KUKA KRL program: cilindro.src, cilindro.dat

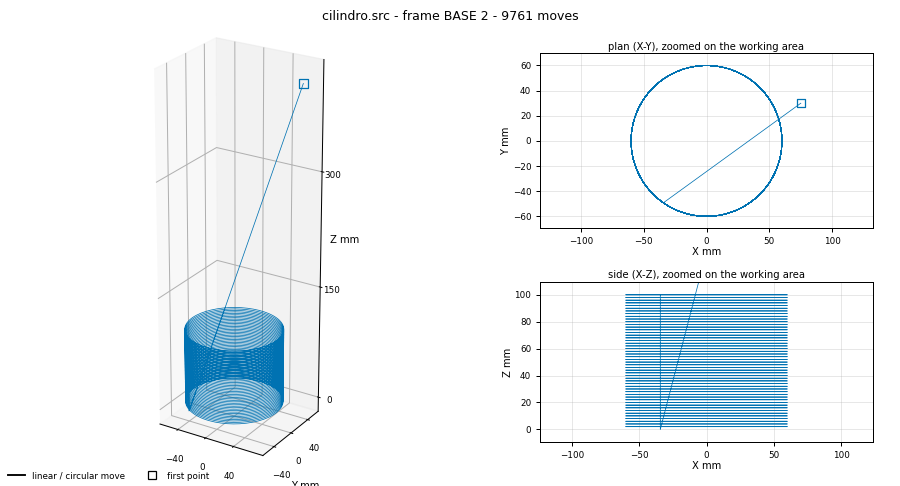
[picture p0: tool path of cilindro.src in frame BASE 2, 9761 of 9763 moves have a stored position in this frame; points joined in program order, loops and branches not executed]
--- cilindro.src ---
&ACCESS RVP
&PARAM TEMPLATE = C:\KRC\Roboter\Template\vorgabe
&PARAM EDITMASK = *
DEF cilindro( )
;FOLD INI;%{PE}%V3.2.0,%MKUKATPBASIS,%CINIT,%VCOMMON,%P
;FOLD BAS INI;%{E}%V3.2.0,%MKUKATPBASIS,%CINIT,%VINIT,%P
GLOBAL INTERRUPT DECL 3 WHEN $STOPMESS==TRUE DO IR_STOPM ( )
INTERRUPT ON 3
BAS (#INITMOV,0 )
;ENDFOLD (BAS INI)
;FOLD A20 INI;%{E}%V3.2.0,%MKUKATPA20,%CINIT,%VINIT,%P
IF ARC20==TRUE THEN
A20 (ARC_INI)
INTERRUPT DECL 6 WHEN $CYCFLAG[3]==FALSE DO A20(TECH_STOP2)
ENDIF
;ENDFOLD (A20 INI)
;FOLD A10 INI;%{E}%V3.2.0,%MKUKATPARC,%CINIT,%VINIT,%P
IF A10_OPTION==#ACTIVE THEN
INTERRUPT DECL 4 WHEN $CYCFLAG[2]==FALSE DO A10 (#APPL_ERROR)
INTERRUPT DECL 7 WHEN A_ARC_SWI==#ACTIVE DO A10 (#ARC_SEAM)
INTERRUPT DECL 5 WHEN A_FLY_ARC==TRUE DO A10 (#HPU_ARC)
INTERRUPT  ON 5
A10_INI ( )
ENDIF
;ENDFOLD (A10 INI)
;FOLD GRIPPER INI;%{E}%V3.2.0,%MKUKATPGRIPPER,%CINIT,%VINIT,%P
USER_GRP(0,DUMMY,DUMMY,GDEFAULT)
;ENDFOLD (GRIPPER INI)
;FOLD SPOT INI;%{E}%V3.2.0,%MKUKATPSPOT,%CINIT,%VINIT,%P
USERSPOT(#INIT)
;ENDFOLD (SPOT INI)
;FOLD TOUCHSENSE INI;%{E}%V3.2.0,%MKUKATPTS,%CINIT,%VINIT,%P
IF H70_OPTION THEN
INTERRUPT DECL 15 WHEN $MEAS_PULSE[TOUCH_I[TOUCH_ACTIVE].IN_NR] DO H70 (6,CD0 )
INTERRUPT DECL 16 WHEN $ZERO_MOVE DO H70 (7,CD0 )
INTERRUPT DECL 17 WHEN $TECHPAR_C[FG_TOUCH,8]>0.5 DO H70 (8,CD0)
H70 (1,CD0 )
ENDIF
;ENDFOLD (TOUCHSENSE INI)
;FOLD USER INI;%{E}%V3.2.0,%MKUKATPUSER,%CINIT,%VINIT,%P
;Make your modifications here
;ENDFOLD (USER INI)
;ENDFOLD (INI)
; SPEED PTP FOR AXIS
$VEL_AXIS[1] = 15
$VEL_AXIS[2] = 15
$VEL_AXIS[3] = 15
$VEL_AXIS[4] = 15
$VEL_AXIS[5] = 15
$VEL_AXIS[6] = 15
;SMOOTHNESS
$APO.CDIS = 2
;ADVANCE
$ADVANCE = 3
;SET TOOL AND BASE
$TOOL = TOOL_DATA[3]
$BASE = BASE_DATA[2]
;HOME
;FOLD PTP HOME Vel=10% DEFAULT
$BWDSTART=FALSE
$H_POS=XHOME
PDAT_ACT=PDEFAULT
FDAT_ACT=FHOME
BAS(#PTP_DAT )
BAS (#VEL_PTP,10 )
PTP XHOME
;ENDFOLD
;USER PROGRAM
;SPEED $VEL.CP
$VEL.CP=0.025
; OUT[TEMP] = 200
; OUT[vent] = 1
; OUT[RPM] = 25
$OUT[1] = TRUE
WAIT SEC 20
$OUT[1] = FALSE
; USER POSES CALLS
PTP {X 75, Y 30, Z 420, A 0, B 90, C 0}
; USER POSES CALLS
LIN {X -34.33, Y -49.21, Z 0.0, A 0, B 90, C 0} C_DIS
WAIT SEC 3
LIN {X -34.33, Y -49.21, Z 2.0, A 0, B 90, C 0} C_DIS
$OUT[1] = TRUE
WAIT SEC 0.8
LIN {X -34.33, Y -49.21, Z 2.0, A 0, B 90, C 0} C_DIS
LIN {X -34.33, Y -49.21, Z 2.0, A 0, B 90, C 0} C_DIS
LIN {X -31.1, Y -51.31, Z 2.0, A 0, B 90, C 0} C_DIS
LIN {X -27.75, Y -53.2, Z 2.0, A 0, B 90, C 0} C_DIS
LIN {X -24.29, Y -54.86, Z 2.0, A 0, B 90, C 0} C_DIS
LIN {X -20.72, Y -56.31, Z 2.0, A 0, B 90, C 0} C_DIS
LIN {X -17.07, Y -57.52, Z 2.0, A 0, B 90, C 0} C_DIS
LIN {X -13.35, Y -58.5, Z 2.0, A 0, B 90, C 0} C_DIS
LIN {X -9.58, Y -59.23, Z 2.0, A 0, B 90, C 0} C_DIS
LIN {X -5.76, Y -59.72, Z 2.0, A 0, B 90, C 0} C_DIS
LIN {X -1.92, Y -59.97, Z 2.0, A 0, B 90, C 0} C_DIS
LIN {X 1.92, Y -59.97, Z 2.0, A 0, B 90, C 0} C_DIS
LIN {X 5.76, Y -59.72, Z 2.0, A 0, B 90, C 0} C_DIS
LIN {X 9.58, Y -59.23, Z 2.0, A 0, B 90, C 0} C_DIS
LIN {X 13.35, Y -58.5, Z 2.0, A 0, B 90, C 0} C_DIS
LIN {X 17.07, Y -57.52, Z 2.0, A 0, B 90, C 0} C_DIS
LIN {X 20.72, Y -56.31, Z 2.0, A 0, B 90, C 0} C_DIS
LIN {X 24.29, Y -54.86, Z 2.0, A 0, B 90, C 0} C_DIS
LIN {X 27.75, Y -53.2, Z 2.0, A 0, B 90, C 0} C_DIS
LIN {X 31.1, Y -51.31, Z 2.0, A 0, B 90, C 0} C_DIS
LIN {X 34.33, Y -49.21, Z 2.0, A 0, B 90, C 0} C_DIS
LIN {X 37.41, Y -46.91, Z 2.0, A 0, B 90, C 0} C_DIS
LIN {X 40.34, Y -44.42, Z 2.0, A 0, B 90, C 0} C_DIS
LIN {X 43.1, Y -41.74, Z 2.0, A 0, B 90, C 0} C_DIS
LIN {X 45.69, Y -38.89, Z 2.0, A 0, B 90, C 0} C_DIS
LIN {X 48.08, Y -35.89, Z 2.0, A 0, B 90, C 0} C_DIS
LIN {X 50.29, Y -32.73, Z 2.0, A 0, B 90, C 0} C_DIS
LIN {X 52.28, Y -29.44, Z 2.0, A 0, B 90, C 0} C_DIS
LIN {X 54.06, Y -26.03, Z 2.0, A 0, B 90, C 0} C_DIS
LIN {X 55.62, Y -22.52, Z 2.0, A 0, B 90, C 0} C_DIS
LIN {X 56.94, Y -18.91, Z 2.0, A 0, B 90, C 0} C_DIS
LIN {X 58.04, Y -15.22, Z 2.0, A 0, B 90, C 0} C_DIS
LIN {X 58.89, Y -11.47, Z 2.0, A 0, B 90, C 0} C_DIS
LIN {X 59.51, Y -7.67, Z 2.0, A 0, B 90, C 0} C_DIS
LIN {X 59.88, Y -3.84, Z 2.0, A 0, B 90, C 0} C_DIS
LIN {X 60.0, Y 0.0, Z 2.0, A 0, B 90, C 0} C_DIS
LIN {X 59.88, Y 3.84, Z 2.0, A 0, B 90, C 0} C_DIS
LIN {X 59.51, Y 7.67, Z 2.0, A 0, B 90, C 0} C_DIS
LIN {X 58.89, Y 11.47, Z 2.0, A 0, B 90, C 0} C_DIS
LIN {X 58.04, Y 15.22, Z 2.0, A 0, B 90, C 0} C_DIS
LIN {X 56.94, Y 18.91, Z 2.0, A 0, B 90, C 0} C_DIS
LIN {X 55.62, Y 22.52, Z 2.0, A 0, B 90, C 0} C_DIS
LIN {X 54.06, Y 26.03, Z 2.0, A 0, B 90, C 0} C_DIS
LIN {X 52.28, Y 29.44, Z 2.0, A 0, B 90, C 0} C_DIS
LIN {X 50.29, Y 32.73, Z 2.0, A 0, B 90, C 0} C_DIS
LIN {X 48.08, Y 35.89, Z 2.0, A 0, B 90, C 0} C_DIS
LIN {X 45.69, Y 38.89, Z 2.0, A 0, B 90, C 0} C_DIS
LIN {X 43.1, Y 41.74, Z 2.0, A 0, B 90, C 0} C_DIS
LIN {X 40.34, Y 44.42, Z 2.0, A 0, B 90, C 0} C_DIS
LIN {X 37.41, Y 46.91, Z 2.0, A 0, B 90, C 0} C_DIS
LIN {X 34.33, Y 49.21, Z 2.0, A 0, B 90, C 0} C_DIS
LIN {X 31.1, Y 51.31, Z 2.0, A 0, B 90, C 0} C_DIS
LIN {X 27.75, Y 53.2, Z 2.0, A 0, B 90, C 0} C_DIS
LIN {X 24.29, Y 54.86, Z 2.0, A 0, B 90, C 0} C_DIS
LIN {X 20.72, Y 56.31, Z 2.0, A 0, B 90, C 0} C_DIS
LIN {X 17.07, Y 57.52, Z 2.0, A 0, B 90, C 0} C_DIS
LIN {X 13.35, Y 58.5, Z 2.0, A 0, B 90, C 0} C_DIS
LIN {X 9.58, Y 59.23, Z 2.0, A 0, B 90, C 0} C_DIS
LIN {X 5.76, Y 59.72, Z 2.0, A 0, B 90, C 0} C_DIS
LIN {X 1.92, Y 59.97, Z 2.0, A 0, B 90, C 0} C_DIS
LIN {X -1.92, Y 59.97, Z 2.0, A 0, B 90, C 0} C_DIS
LIN {X -5.76, Y 59.72, Z 2.0, A 0, B 90, C 0} C_DIS
LIN {X -9.58, Y 59.23, Z 2.0, A 0, B 90, C 0} C_DIS
LIN {X -13.35, Y 58.5, Z 2.0, A 0, B 90, C 0} C_DIS
LIN {X -17.07, Y 57.52, Z 2.0, A 0, B 90, C 0} C_DIS
LIN {X -20.72, Y 56.31, Z 2.0, A 0, B 90, C 0} C_DIS
LIN {X -24.29, Y 54.86, Z 2.0, A 0, B 90, C 0} C_DIS
LIN {X -27.75, Y 53.2, Z 2.0, A 0, B 90, C 0} C_DIS
LIN {X -31.1, Y 51.31, Z 2.0, A 0, B 90, C 0} C_DIS
LIN {X -34.33, Y 49.21, Z 2.0, A 0, B 90, C 0} C_DIS
LIN {X -37.41, Y 46.91, Z 2.0, A 0, B 90, C 0} C_DIS
LIN {X -40.34, Y 44.42, Z 2.0, A 0, B 90, C 0} C_DIS
LIN {X -43.1, Y 41.74, Z 2.0, A 0, B 90, C 0} C_DIS
LIN {X -45.69, Y 38.89, Z 2.0, A 0, B 90, C 0} C_DIS
LIN {X -48.08, Y 35.89, Z 2.0, A 0, B 90, C 0} C_DIS
LIN {X -50.29, Y 32.73, Z 2.0, A 0, B 90, C 0} C_DIS
LIN {X -52.28, Y 29.44, Z 2.0, A 0, B 90, C 0} C_DIS
LIN {X -54.06, Y 26.03, Z 2.0, A 0, B 90, C 0} C_DIS
LIN {X -55.62, Y 22.52, Z 2.0, A 0, B 90, C 0} C_DIS
LIN {X -56.94, Y 18.91, Z 2.0, A 0, B 90, C 0} C_DIS
LIN {X -58.04, Y 15.22, Z 2.0, A 0, B 90, C 0} C_DIS
LIN {X -58.89, Y 11.47, Z 2.0, A 0, B 90, C 0} C_DIS
LIN {X -59.51, Y 7.67, Z 2.0, A 0, B 90, C 0} C_DIS
LIN {X -59.88, Y 3.84, Z 2.0, A 0, B 90, C 0} C_DIS
LIN {X -60.0, Y -0.0, Z 2.0, A 0, B 90, C 0} C_DIS
LIN {X -59.88, Y -3.84, Z 2.0, A 0, B 90, C 0} C_DIS
LIN {X -59.51, Y -7.67, Z 2.0, A 0, B 90, C 0} C_DIS
LIN {X -58.89, Y -11.47, Z 2.0, A 0, B 90, C 0} C_DIS
LIN {X -58.04, Y -15.22, Z 2.0, A 0, B 90, C 0} C_DIS
LIN {X -56.94, Y -18.91, Z 2.0, A 0, B 90, C 0} C_DIS
LIN {X -55.62, Y -22.52, Z 2.0, A 0, B 90, C 0} C_DIS
LIN {X -54.06, Y -26.03, Z 2.0, A 0, B 90, C 0} C_DIS
LIN {X -52.28, Y -29.44, Z 2.0, A 0, B 90, C 0} C_DIS
LIN {X -50.29, Y -32.73, Z 2.0, A 0, B 90, C 0} C_DIS
LIN {X -48.08, Y -35.89, Z 2.0, A 0, B 90, C 0} C_DIS
LIN {X -45.69, Y -38.89, Z 2.0, A 0, B 90, C 0} C_DIS
LIN {X -43.1, Y -41.74, Z 2.0, A 0, B 90, C 0} C_DIS
LIN {X -40.34, Y -44.42, Z 2.0, A 0, B 90, C 0} C_DIS
LIN {X -37.41, Y -46.91, Z 2.0, A 0, B 90, C 0} C_DIS
LIN {X -37.13, Y -47.12, Z 2.0, A 0, B 90, C 0} C_DIS
$OUT[1] = FALSE

; END LAYER 0
LIN {X -34.33, Y -49.21, Z 2.0, A 0, B 90, C 0} C_DIS
WAIT SEC 3
LIN {X -34.33, Y -49.21, Z 4.0, A 0, B 90, C 0} C_DIS
$OUT[1] = TRUE
WAIT SEC 0.8
LIN {X -34.33, Y -49.21, Z 4.0, A 0, B 90, C 0} C_DIS
LIN {X -34.33, Y -49.21, Z 4.0, A 0, B 90, C 0} C_DIS
LIN {X -34.2, Y -49.29, Z 4.0, A 0, B 90, C 0} C_DIS
LIN {X -31.1, Y -51.31, Z 4.0, A 0, B 90, C 0} C_DIS
LIN {X -30.97, Y -51.38, Z 4.0, A 0, B 90, C 0} C_DIS
LIN {X -27.75, Y -53.2, Z 4.0, A 0, B 90, C 0} C_DIS
LIN {X -27.61, Y -53.26, Z 4.0, A 0, B 90, C 0} C_DIS
LIN {X -24.29, Y -54.86, Z 4.0, A 0, B 90, C 0} C_DIS
LIN {X -24.14, Y -54.92, Z 4.0, A 0, B 90, C 0} C_DIS
LIN {X -20.72, Y -56.31, Z 4.0, A 0, B 90, C 0} C_DIS
LIN {X -20.58, Y -56.36, Z 4.0, A 0, B 90, C 0} C_DIS
LIN {X -17.07, Y -57.52, Z 4.0, A 0, B 90, C 0} C_DIS
LIN {X -16.92, Y -57.56, Z 4.0, A 0, B 90, C 0} C_DIS
LIN {X -13.35, Y -58.5, Z 4.0, A 0, B 90, C 0} C_DIS
LIN {X -13.2, Y -58.53, Z 4.0, A 0, B 90, C 0} C_DIS
LIN {X -9.58, Y -59.23, Z 4.0, A 0, B 90, C 0} C_DIS
LIN {X -9.42, Y -59.25, Z 4.0, A 0, B 90, C 0} C_DIS
LIN {X -5.76, Y -59.72, Z 4.0, A 0, B 90, C 0} C_DIS
LIN {X -5.61, Y -59.73, Z 4.0, A 0, B 90, C 0} C_DIS
LIN {X -1.92, Y -59.97, Z 4.0, A 0, B 90, C 0} C_DIS
LIN {X -1.77, Y -59.97, Z 4.0, A 0, B 90, C 0} C_DIS
LIN {X 1.92, Y -59.97, Z 4.0, A 0, B 90, C 0} C_DIS
LIN {X 2.08, Y -59.96, Z 4.0, A 0, B 90, C 0} C_DIS
LIN {X 5.76, Y -59.72, Z 4.0, A 0, B 90, C 0} C_DIS
LIN {X 5.91, Y -59.7, Z 4.0, A 0, B 90, C 0} C_DIS
LIN {X 9.58, Y -59.23, Z 4.0, A 0, B 90, C 0} C_DIS
LIN {X 9.73, Y -59.2, Z 4.0, A 0, B 90, C 0} C_DIS
LIN {X 13.35, Y -58.5, Z 4.0, A 0, B 90, C 0} C_DIS
LIN {X 13.5, Y -58.46, Z 4.0, A 0, B 90, C 0} C_DIS
LIN {X 17.07, Y -57.52, Z 4.0, A 0, B 90, C 0} C_DIS
LIN {X 17.22, Y -57.47, Z 4.0, A 0, B 90, C 0} C_DIS
LIN {X 20.72, Y -56.31, Z 4.0, A 0, B 90, C 0} C_DIS
LIN {X 20.86, Y -56.25, Z 4.0, A 0, B 90, C 0} C_DIS
LIN {X 24.29, Y -54.86, Z 4.0, A 0, B 90, C 0} C_DIS
LIN {X 24.43, Y -54.8, Z 4.0, A 0, B 90, C 0} C_DIS
LIN {X 27.75, Y -53.2, Z 4.0, A 0, B 90, C 0} C_DIS
LIN {X 27.89, Y -53.12, Z 4.0, A 0, B 90, C 0} C_DIS
LIN {X 31.1, Y -51.31, Z 4.0, A 0, B 90, C 0} C_DIS
LIN {X 31.23, Y -51.22, Z 4.0, A 0, B 90, C 0} C_DIS
LIN {X 34.33, Y -49.21, Z 4.0, A 0, B 90, C 0} C_DIS
LIN {X 34.45, Y -49.12, Z 4.0, A 0, B 90, C 0} C_DIS
LIN {X 37.41, Y -46.91, Z 4.0, A 0, B 90, C 0} C_DIS
LIN {X 37.53, Y -46.81, Z 4.0, A 0, B 90, C 0} C_DIS
LIN {X 40.34, Y -44.42, Z 4.0, A 0, B 90, C 0} C_DIS
LIN {X 40.45, Y -44.31, Z 4.0, A 0, B 90, C 0} C_DIS
LIN {X 43.1, Y -41.74, Z 4.0, A 0, B 90, C 0} C_DIS
LIN {X 43.2, Y -41.63, Z 4.0, A 0, B 90, C 0} C_DIS
LIN {X 45.69, Y -38.89, Z 4.0, A 0, B 90, C 0} C_DIS
LIN {X 45.78, Y -38.77, Z 4.0, A 0, B 90, C 0} C_DIS
LIN {X 48.08, Y -35.89, Z 4.0, A 0, B 90, C 0} C_DIS
LIN {X 48.17, Y -35.76, Z 4.0, A 0, B 90, C 0} C_DIS
LIN {X 50.29, Y -32.73, Z 4.0, A 0, B 90, C 0} C_DIS
LIN {X 50.37, Y -32.6, Z 4.0, A 0, B 90, C 0} C_DIS
LIN {X 52.28, Y -29.44, Z 4.0, A 0, B 90, C 0} C_DIS
LIN {X 52.35, Y -29.31, Z 4.0, A 0, B 90, C 0} C_DIS
LIN {X 54.06, Y -26.03, Z 4.0, A 0, B 90, C 0} C_DIS
LIN {X 54.12, Y -25.89, Z 4.0, A 0, B 90, C 0} C_DIS
LIN {X 55.62, Y -22.52, Z 4.0, A 0, B 90, C 0} C_DIS
LIN {X 55.67, Y -22.37, Z 4.0, A 0, B 90, C 0} C_DIS
LIN {X 56.94, Y -18.91, Z 4.0, A 0, B 90, C 0} C_DIS
LIN {X 56.99, Y -18.76, Z 4.0, A 0, B 90, C 0} C_DIS
LIN {X 58.04, Y -15.22, Z 4.0, A 0, B 90, C 0} C_DIS
LIN {X 58.07, Y -15.07, Z 4.0, A 0, B 90, C 0} C_DIS
LIN {X 58.89, Y -11.47, Z 4.0, A 0, B 90, C 0} C_DIS
LIN {X 58.92, Y -11.32, Z 4.0, A 0, B 90, C 0} C_DIS
LIN {X 59.51, Y -7.67, Z 4.0, A 0, B 90, C 0} C_DIS
LIN {X 59.52, Y -7.52, Z 4.0, A 0, B 90, C 0} C_DIS
LIN {X 59.88, Y -3.84, Z 4.0, A 0, B 90, C 0} C_DIS
LIN {X 59.88, Y -3.69, Z 4.0, A 0, B 90, C 0} C_DIS
LIN {X 60.0, Y 0.0, Z 4.0, A 0, B 90, C 0} C_DIS
LIN {X 60.0, Y 0.15, Z 4.0, A 0, B 90, C 0} C_DIS
LIN {X 59.88, Y 3.84, Z 4.0, A 0, B 90, C 0} C_DIS
LIN {X 59.86, Y 4.0, Z 4.0, A 0, B 90, C 0} C_DIS
LIN {X 59.51, Y 7.67, Z 4.0, A 0, B 90, C 0} C_DIS
LIN {X 59.48, Y 7.82, Z 4.0, A 0, B 90, C 0} C_DIS
LIN {X 58.89, Y 11.47, Z 4.0, A 0, B 90, C 0} C_DIS
LIN {X 58.86, Y 11.62, Z 4.0, A 0, B 90, C 0} C_DIS
LIN {X 58.04, Y 15.22, Z 4.0, A 0, B 90, C 0} C_DIS
LIN {X 57.99, Y 15.37, Z 4.0, A 0, B 90, C 0} C_DIS
LIN {X 56.94, Y 18.91, Z 4.0, A 0, B 90, C 0} C_DIS
LIN {X 56.89, Y 19.05, Z 4.0, A 0, B 90, C 0} C_DIS
LIN {X 55.62, Y 22.52, Z 4.0, A 0, B 90, C 0} C_DIS
LIN {X 55.55, Y 22.66, Z 4.0, A 0, B 90, C 0} C_DIS
LIN {X 54.06, Y 26.03, Z 4.0, A 0, B 90, C 0} C_DIS
LIN {X 53.99, Y 26.17, Z 4.0, A 0, B 90, C 0} C_DIS
LIN {X 52.28, Y 29.44, Z 4.0, A 0, B 90, C 0} C_DIS
LIN {X 52.2, Y 29.57, Z 4.0, A 0, B 90, C 0} C_DIS
LIN {X 50.29, Y 32.73, Z 4.0, A 0, B 90, C 0} C_DIS
LIN {X 50.2, Y 32.86, Z 4.0, A 0, B 90, C 0} C_DIS
LIN {X 48.08, Y 35.89, Z 4.0, A 0, B 90, C 0} C_DIS
LIN {X 47.99, Y 36.01, Z 4.0, A 0, B 90, C 0} C_DIS
LIN {X 45.69, Y 38.89, Z 4.0, A 0, B 90, C 0} C_DIS
LIN {X 45.58, Y 39.01, Z 4.0, A 0, B 90, C 0} C_DIS
LIN {X 43.1, Y 41.74, Z 4.0, A 0, B 90, C 0} C_DIS
LIN {X 42.99, Y 41.85, Z 4.0, A 0, B 90, C 0} C_DIS
LIN {X 40.34, Y 44.42, Z 4.0, A 0, B 90, C 0} C_DIS
LIN {X 40.22, Y 44.52, Z 4.0, A 0, B 90, C 0} C_DIS
LIN {X 37.41, Y 46.91, Z 4.0, A 0, B 90, C 0} C_DIS
LIN {X 37.29, Y 47.0, Z 4.0, A 0, B 90, C 0} C_DIS
LIN {X 34.33, Y 49.21, Z 4.0, A 0, B 90, C 0} C_DIS
LIN {X 34.2, Y 49.29, Z 4.0, A 0, B 90, C 0} C_DIS
LIN {X 31.1, Y 51.31, Z 4.0, A 0, B 90, C 0} C_DIS
LIN {X 30.97, Y 51.38, Z 4.0, A 0, B 90, C 0} C_DIS
LIN {X 27.75, Y 53.2, Z 4.0, A 0, B 90, C 0} C_DIS
LIN {X 27.61, Y 53.26, Z 4.0, A 0, B 90, C 0} C_DIS
LIN {X 24.29, Y 54.86, Z 4.0, A 0, B 90, C 0} C_DIS
LIN {X 24.14, Y 54.92, Z 4.0, A 0, B 90, C 0} C_DIS
LIN {X 20.72, Y 56.31, Z 4.0, A 0, B 90, C 0} C_DIS
LIN {X 20.58, Y 56.36, Z 4.0, A 0, B 90, C 0} C_DIS
LIN {X 17.07, Y 57.52, Z 4.0, A 0, B 90, C 0} C_DIS
LIN {X 16.92, Y 57.56, Z 4.0, A 0, B 90, C 0} C_DIS
LIN {X 13.35, Y 58.5, Z 4.0, A 0, B 90, C 0} C_DIS
LIN {X 13.2, Y 58.53, Z 4.0, A 0, B 90, C 0} C_DIS
LIN {X 9.58, Y 59.23, Z 4.0, A 0, B 90, C 0} C_DIS
LIN {X 9.42, Y 59.25, Z 4.0, A 0, B 90, C 0} C_DIS
LIN {X 5.76, Y 59.72, Z 4.0, A 0, B 90, C 0} C_DIS
LIN {X 5.61, Y 59.73, Z 4.0, A 0, B 90, C 0} C_DIS
LIN {X 1.92, Y 59.97, Z 4.0, A 0, B 90, C 0} C_DIS
LIN {X 1.77, Y 59.97, Z 4.0, A 0, B 90, C 0} C_DIS
LIN {X -1.92, Y 59.97, Z 4.0, A 0, B 90, C 0} C_DIS
LIN {X -2.08, Y 59.96, Z 4.0, A 0, B 90, C 0} C_DIS
LIN {X -5.76, Y 59.72, Z 4.0, A 0, B 90, C 0} C_DIS
LIN {X -5.91, Y 59.7, Z 4.0, A 0, B 90, C 0} C_DIS
LIN {X -9.58, Y 59.23, Z 4.0, A 0, B 90, C 0} C_DIS
LIN {X -9.73, Y 59.2, Z 4.0, A 0, B 90, C 0} C_DIS
LIN {X -13.35, Y 58.5, Z 4.0, A 0, B 90, C 0} C_DIS
LIN {X -13.5, Y 58.46, Z 4.0, A 0, B 90, C 0} C_DIS
LIN {X -17.07, Y 57.52, Z 4.0, A 0, B 90, C 0} C_DIS
LIN {X -17.22, Y 57.47, Z 4.0, A 0, B 90, C 0} C_DIS
LIN {X -20.72, Y 56.31, Z 4.0, A 0, B 90, C 0} C_DIS
LIN {X -20.86, Y 56.25, Z 4.0, A 0, B 90, C 0} C_DIS
LIN {X -24.29, Y 54.86, Z 4.0, A 0, B 90, C 0} C_DIS
LIN {X -24.43, Y 54.8, Z 4.0, A 0, B 90, C 0} C_DIS
LIN {X -27.75, Y 53.2, Z 4.0, A 0, B 90, C 0} C_DIS
LIN {X -27.89, Y 53.12, Z 4.0, A 0, B 90, C 0} C_DIS
LIN {X -31.1, Y 51.31, Z 4.0, A 0, B 90, C 0} C_DIS
LIN {X -31.23, Y 51.22, Z 4.0, A 0, B 90, C 0} C_DIS
LIN {X -34.33, Y 49.21, Z 4.0, A 0, B 90, C 0} C_DIS
LIN {X -34.45, Y 49.12, Z 4.0, A 0, B 90, C 0} C_DIS
LIN {X -37.41, Y 46.91, Z 4.0, A 0, B 90, C 0} C_DIS
LIN {X -37.53, Y 46.81, Z 4.0, A 0, B 90, C 0} C_DIS
LIN {X -40.34, Y 44.42, Z 4.0, A 0, B 90, C 0} C_DIS
LIN {X -40.45, Y 44.31, Z 4.0, A 0, B 90, C 0} C_DIS
LIN {X -43.1, Y 41.74, Z 4.0, A 0, B 90, C 0} C_DIS
LIN {X -43.2, Y 41.63, Z 4.0, A 0, B 90, C 0} C_DIS
LIN {X -45.69, Y 38.89, Z 4.0, A 0, B 90, C 0} C_DIS
LIN {X -45.78, Y 38.77, Z 4.0, A 0, B 90, C 0} C_DIS
LIN {X -48.08, Y 35.89, Z 4.0, A 0, B 90, C 0} C_DIS
LIN {X -48.17, Y 35.76, Z 4.0, A 0, B 90, C 0} C_DIS
LIN {X -50.29, Y 32.73, Z 4.0, A 0, B 90, C 0} C_DIS
LIN {X -50.37, Y 32.6, Z 4.0, A 0, B 90, C 0} C_DIS
LIN {X -52.28, Y 29.44, Z 4.0, A 0, B 90, C 0} C_DIS
LIN {X -52.35, Y 29.31, Z 4.0, A 0, B 90, C 0} C_DIS
LIN {X -54.06, Y 26.03, Z 4.0, A 0, B 90, C 0} C_DIS
LIN {X -54.12, Y 25.89, Z 4.0, A 0, B 90, C 0} C_DIS
LIN {X -55.62, Y 22.52, Z 4.0, A 0, B 90, C 0} C_DIS
LIN {X -55.67, Y 22.37, Z 4.0, A 0, B 90, C 0} C_DIS
LIN {X -56.94, Y 18.91, Z 4.0, A 0, B 90, C 0} C_DIS
LIN {X -56.99, Y 18.76, Z 4.0, A 0, B 90, C 0} C_DIS
LIN {X -58.04, Y 15.22, Z 4.0, A 0, B 90, C 0} C_DIS
LIN {X -58.07, Y 15.07, Z 4.0, A 0, B 90, C 0} C_DIS
LIN {X -58.89, Y 11.47, Z 4.0, A 0, B 90, C 0} C_DIS
LIN {X -58.92, Y 11.32, Z 4.0, A 0, B 90, C 0} C_DIS
LIN {X -59.51, Y 7.67, Z 4.0, A 0, B 90, C 0} C_DIS
LIN {X -59.52, Y 7.52, Z 4.0, A 0, B 90, C 0} C_DIS
LIN {X -59.88, Y 3.84, Z 4.0, A 0, B 90, C 0} C_DIS
LIN {X -59.88, Y 3.69, Z 4.0, A 0, B 90, C 0} C_DIS
LIN {X -60.0, Y -0.0, Z 4.0, A 0, B 90, C 0} C_DIS
LIN {X -60.0, Y -0.15, Z 4.0, A 0, B 90, C 0} C_DIS
LIN {X -59.88, Y -3.84, Z 4.0, A 0, B 90, C 0} C_DIS
LIN {X -59.86, Y -4.0, Z 4.0, A 0, B 90, C 0} C_DIS
LIN {X -59.51, Y -7.67, Z 4.0, A 0, B 90, C 0} C_DIS
LIN {X -59.48, Y -7.82, Z 4.0, A 0, B 90, C 0} C_DIS
LIN {X -58.89, Y -11.47, Z 4.0, A 0, B 90, C 0} C_DIS
LIN {X -58.86, Y -11.62, Z 4.0, A 0, B 90, C 0} C_DIS
LIN {X -58.04, Y -15.22, Z 4.0, A 0, B 90, C 0} C_DIS
LIN {X -57.99, Y -15.37, Z 4.0, A 0, B 90, C 0} C_DIS
LIN {X -56.94, Y -18.91, Z 4.0, A 0, B 90, C 0} C_DIS
LIN {X -56.89, Y -19.05, Z 4.0, A 0, B 90, C 0} C_DIS
LIN {X -55.62, Y -22.52, Z 4.0, A 0, B 90, C 0} C_DIS
LIN {X -55.55, Y -22.66, Z 4.0, A 0, B 90, C 0} C_DIS
LIN {X -54.06, Y -26.03, Z 4.0, A 0, B 90, C 0} C_DIS
LIN {X -53.99, Y -26.17, Z 4.0, A 0, B 90, C 0} C_DIS
LIN {X -52.28, Y -29.44, Z 4.0, A 0, B 90, C 0} C_DIS
LIN {X -52.2, Y -29.57, Z 4.0, A 0, B 90, C 0} C_DIS
LIN {X -50.29, Y -32.73, Z 4.0, A 0, B 90, C 0} C_DIS
LIN {X -50.2, Y -32.86, Z 4.0, A 0, B 90, C 0} C_DIS
LIN {X -48.08, Y -35.89, Z 4.0, A 0, B 90, C 0} C_DIS
LIN {X -47.99, Y -36.01, Z 4.0, A 0, B 90, C 0} C_DIS
LIN {X -45.69, Y -38.89, Z 4.0, A 0, B 90, C 0} C_DIS
LIN {X -45.58, Y -39.01, Z 4.0, A 0, B 90, C 0} C_DIS
LIN {X -43.1, Y -41.74, Z 4.0, A 0, B 90, C 0} C_DIS
LIN {X -42.99, Y -41.85, Z 4.0, A 0, B 90, C 0} C_DIS
LIN {X -40.34, Y -44.42, Z 4.0, A 0, B 90, C 0} C_DIS
LIN {X -40.22, Y -44.52, Z 4.0, A 0, B 90, C 0} C_DIS
LIN {X -37.41, Y -46.91, Z 4.0, A 0, B 90, C 0} C_DIS
LIN {X -37.29, Y -47.0, Z 4.0, A 0, B 90, C 0} C_DIS
LIN {X -37.13, Y -47.12, Z 4.0, A 0, B 90, C 0} C_DIS
$OUT[1] = FALSE

; END LAYER 1
LIN {X -34.33, Y -49.21, Z 4.0, A 0, B 90, C 0} C_DIS
WAIT SEC 3
LIN {X -34.33, Y -49.21, Z 6.0, A 0, B 90, C 0} C_DIS
$OUT[1] = TRUE
WAIT SEC 0.8
LIN {X -34.33, Y -49.21, Z 6.0, A 0, B 90, C 0} C_DIS
LIN {X -34.33, Y -49.21, Z 6.0, A 0, B 90, C 0} C_DIS
LIN {X -34.07, Y -49.38, Z 6.0, A 0, B 90, C 0} C_DIS
LIN {X -31.1, Y -51.31, Z 6.0, A 0, B 90, C 0} C_DIS
LIN {X -30.84, Y -51.46, Z 6.0, A 0, B 90, C 0} C_DIS
LIN {X -27.75, Y -53.2, Z 6.0, A 0, B 90, C 0} C_DIS
LIN {X -27.48, Y -53.33, Z 6.0, A 0, B 90, C 0} C_DIS
LIN {X -24.29, Y -54.86, Z 6.0, A 0, B 90, C 0} C_DIS
LIN {X -24.0, Y -54.98, Z 6.0, A 0, B 90, C 0} C_DIS
LIN {X -20.72, Y -56.31, Z 6.0, A 0, B 90, C 0} C_DIS
LIN {X -20.43, Y -56.41, Z 6.0, A 0, B 90, C 0} C_DIS
LIN {X -17.07, Y -57.52, Z 6.0, A 0, B 90, C 0} C_DIS
LIN {X -16.77, Y -57.6, Z 6.0, A 0, B 90, C 0} C_DIS
LIN {X -13.35, Y -58.5, Z 6.0, A 0, B 90, C 0} C_DIS
LIN {X -13.05, Y -58.55, Z 6.0, A 0, B 90, C 0} C_DIS
LIN {X -9.58, Y -59.23, Z 6.0, A 0, B 90, C 0} C_DIS
LIN {X -9.27, Y -59.27, Z 6.0, A 0, B 90, C 0} C_DIS
LIN {X -5.76, Y -59.72, Z 6.0, A 0, B 90, C 0} C_DIS
LIN {X -5.45, Y -59.74, Z 6.0, A 0, B 90, C 0} C_DIS
LIN {X -1.92, Y -59.97, Z 6.0, A 0, B 90, C 0} C_DIS
LIN {X -1.62, Y -59.97, Z 6.0, A 0, B 90, C 0} C_DIS
LIN {X 1.92, Y -59.97, Z 6.0, A 0, B 90, C 0} C_DIS
LIN {X 2.23, Y -59.95, Z 6.0, A 0, B 90, C 0} C_DIS
LIN {X 5.76, Y -59.72, Z 6.0, A 0, B 90, C 0} C_DIS
LIN {X 6.07, Y -59.68, Z 6.0, A 0, B 90, C 0} C_DIS
LIN {X 9.58, Y -59.23, Z 6.0, A 0, B 90, C 0} C_DIS
LIN {X 9.88, Y -59.17, Z 6.0, A 0, B 90, C 0} C_DIS
LIN {X 13.35, Y -58.5, Z 6.0, A 0, B 90, C 0} C_DIS
LIN {X 13.65, Y -58.42, Z 6.0, A 0, B 90, C 0} C_DIS
LIN {X 17.07, Y -57.52, Z 6.0, A 0, B 90, C 0} C_DIS
LIN {X 17.36, Y -57.42, Z 6.0, A 0, B 90, C 0} C_DIS
LIN {X 20.72, Y -56.31, Z 6.0, A 0, B 90, C 0} C_DIS
LIN {X 21.01, Y -56.19, Z 6.0, A 0, B 90, C 0} C_DIS
LIN {X 24.29, Y -54.86, Z 6.0, A 0, B 90, C 0} C_DIS
LIN {X 24.56, Y -54.73, Z 6.0, A 0, B 90, C 0} C_DIS
LIN {X 27.75, Y -53.2, Z 6.0, A 0, B 90, C 0} C_DIS
LIN {X 28.02, Y -53.04, Z 6.0, A 0, B 90, C 0} C_DIS
LIN {X 31.1, Y -51.31, Z 6.0, A 0, B 90, C 0} C_DIS
LIN {X 31.36, Y -51.14, Z 6.0, A 0, B 90, C 0} C_DIS
LIN {X 34.33, Y -49.21, Z 6.0, A 0, B 90, C 0} C_DIS
LIN {X 34.57, Y -49.03, Z 6.0, A 0, B 90, C 0} C_DIS
LIN {X 37.41, Y -46.91, Z 6.0, A 0, B 90, C 0} C_DIS
LIN {X 37.64, Y -46.71, Z 6.0, A 0, B 90, C 0} C_DIS
LIN {X 40.34, Y -44.42, Z 6.0, A 0, B 90, C 0} C_DIS
LIN {X 40.56, Y -44.2, Z 6.0, A 0, B 90, C 0} C_DIS
LIN {X 43.1, Y -41.74, Z 6.0, A 0, B 90, C 0} C_DIS
LIN {X 43.31, Y -41.51, Z 6.0, A 0, B 90, C 0} C_DIS
LIN {X 45.69, Y -38.89, Z 6.0, A 0, B 90, C 0} C_DIS
LIN {X 45.88, Y -38.65, Z 6.0, A 0, B 90, C 0} C_DIS
LIN {X 48.08, Y -35.89, Z 6.0, A 0, B 90, C 0} C_DIS
LIN {X 48.26, Y -35.63, Z 6.0, A 0, B 90, C 0} C_DIS
LIN {X 50.29, Y -32.73, Z 6.0, A 0, B 90, C 0} C_DIS
LIN {X 50.44, Y -32.47, Z 6.0, A 0, B 90, C 0} C_DIS
LIN {X 52.28, Y -29.44, Z 6.0, A 0, B 90, C 0} C_DIS
LIN {X 52.42, Y -29.17, Z 6.0, A 0, B 90, C 0} C_DIS
LIN {X 54.06, Y -26.03, Z 6.0, A 0, B 90, C 0} C_DIS
LIN {X 54.18, Y -25.75, Z 6.0, A 0, B 90, C 0} C_DIS
LIN {X 55.62, Y -22.52, Z 6.0, A 0, B 90, C 0} C_DIS
LIN {X 55.72, Y -22.23, Z 6.0, A 0, B 90, C 0} C_DIS
LIN {X 56.94, Y -18.91, Z 6.0, A 0, B 90, C 0} C_DIS
LIN {X 57.03, Y -18.61, Z 6.0, A 0, B 90, C 0} C_DIS
LIN {X 58.04, Y -15.22, Z 6.0, A 0, B 90, C 0} C_DIS
LIN {X 58.11, Y -14.92, Z 6.0, A 0, B 90, C 0} C_DIS
LIN {X 58.89, Y -11.47, Z 6.0, A 0, B 90, C 0} C_DIS
LIN {X 58.94, Y -11.17, Z 6.0, A 0, B 90, C 0} C_DIS
LIN {X 59.51, Y -7.67, Z 6.0, A 0, B 90, C 0} C_DIS
LIN {X 59.54, Y -7.37, Z 6.0, A 0, B 90, C 0} C_DIS
LIN {X 59.88, Y -3.84, Z 6.0, A 0, B 90, C 0} C_DIS
LIN {X 59.89, Y -3.54, Z 6.0, A 0, B 90, C 0} C_DIS
LIN {X 60.0, Y 0.0, Z 6.0, A 0, B 90, C 0} C_DIS
LIN {X 59.99, Y 0.31, Z 6.0, A 0, B 90, C 0} C_DIS
LIN {X 59.88, Y 3.84, Z 6.0, A 0, B 90, C 0} C_DIS
LIN {X 59.85, Y 4.15, Z 6.0, A 0, B 90, C 0} C_DIS
LIN {X 59.51, Y 7.67, Z 6.0, A 0, B 90, C 0} C_DIS
LIN {X 59.46, Y 7.98, Z 6.0, A 0, B 90, C 0} C_DIS
LIN {X 58.89, Y 11.47, Z 6.0, A 0, B 90, C 0} C_DIS
LIN {X 58.83, Y 11.77, Z 6.0, A 0, B 90, C 0} C_DIS
LIN {X 58.04, Y 15.22, Z 6.0, A 0, B 90, C 0} C_DIS
LIN {X 57.95, Y 15.51, Z 6.0, A 0, B 90, C 0} C_DIS
LIN {X 56.94, Y 18.91, Z 6.0, A 0, B 90, C 0} C_DIS
LIN {X 56.84, Y 19.2, Z 6.0, A 0, B 90, C 0} C_DIS
LIN {X 55.62, Y 22.52, Z 6.0, A 0, B 90, C 0} C_DIS
LIN {X 55.49, Y 22.8, Z 6.0, A 0, B 90, C 0} C_DIS
LIN {X 54.06, Y 26.03, Z 6.0, A 0, B 90, C 0} C_DIS
LIN {X 53.92, Y 26.31, Z 6.0, A 0, B 90, C 0} C_DIS
LIN {X 52.28, Y 29.44, Z 6.0, A 0, B 90, C 0} C_DIS
LIN {X 52.12, Y 29.71, Z 6.0, A 0, B 90, C 0} C_DIS
LIN {X 50.29, Y 32.73, Z 6.0, A 0, B 90, C 0} C_DIS
LIN {X 50.11, Y 32.98, Z 6.0, A 0, B 90, C 0} C_DIS
LIN {X 48.08, Y 35.89, Z 6.0, A 0, B 90, C 0} C_DIS
LIN {X 47.89, Y 36.13, Z 6.0, A 0, B 90, C 0} C_DIS
LIN {X 45.69, Y 38.89, Z 6.0, A 0, B 90, C 0} C_DIS
LIN {X 45.48, Y 39.12, Z 6.0, A 0, B 90, C 0} C_DIS
LIN {X 43.1, Y 41.74, Z 6.0, A 0, B 90, C 0} C_DIS
LIN {X 42.88, Y 41.96, Z 6.0, A 0, B 90, C 0} C_DIS
LIN {X 40.34, Y 44.42, Z 6.0, A 0, B 90, C 0} C_DIS
LIN {X 40.1, Y 44.62, Z 6.0, A 0, B 90, C 0} C_DIS
LIN {X 37.41, Y 46.91, Z 6.0, A 0, B 90, C 0} C_DIS
LIN {X 37.16, Y 47.09, Z 6.0, A 0, B 90, C 0} C_DIS
LIN {X 34.33, Y 49.21, Z 6.0, A 0, B 90, C 0} C_DIS
LIN {X 34.07, Y 49.38, Z 6.0, A 0, B 90, C 0} C_DIS
LIN {X 31.1, Y 51.31, Z 6.0, A 0, B 90, C 0} C_DIS
LIN {X 30.84, Y 51.46, Z 6.0, A 0, B 90, C 0} C_DIS
LIN {X 27.75, Y 53.2, Z 6.0, A 0, B 90, C 0} C_DIS
LIN {X 27.48, Y 53.33, Z 6.0, A 0, B 90, C 0} C_DIS
LIN {X 24.29, Y 54.86, Z 6.0, A 0, B 90, C 0} C_DIS
LIN {X 24.0, Y 54.98, Z 6.0, A 0, B 90, C 0} C_DIS
LIN {X 20.72, Y 56.31, Z 6.0, A 0, B 90, C 0} C_DIS
LIN {X 20.43, Y 56.41, Z 6.0, A 0, B 90, C 0} C_DIS
LIN {X 17.07, Y 57.52, Z 6.0, A 0, B 90, C 0} C_DIS
LIN {X 16.77, Y 57.6, Z 6.0, A 0, B 90, C 0} C_DIS
LIN {X 13.35, Y 58.5, Z 6.0, A 0, B 90, C 0} C_DIS
LIN {X 13.05, Y 58.55, Z 6.0, A 0, B 90, C 0} C_DIS
LIN {X 9.58, Y 59.23, Z 6.0, A 0, B 90, C 0} C_DIS
LIN {X 9.27, Y 59.27, Z 6.0, A 0, B 90, C 0} C_DIS
LIN {X 5.76, Y 59.72, Z 6.0, A 0, B 90, C 0} C_DIS
LIN {X 5.45, Y 59.74, Z 6.0, A 0, B 90, C 0} C_DIS
LIN {X 1.92, Y 59.97, Z 6.0, A 0, B 90, C 0} C_DIS
LIN {X 1.62, Y 59.97, Z 6.0, A 0, B 90, C 0} C_DIS
LIN {X -1.92, Y 59.97, Z 6.0, A 0, B 90, C 0} C_DIS
LIN {X -2.23, Y 59.95, Z 6.0, A 0, B 90, C 0} C_DIS
LIN {X -5.76, Y 59.72, Z 6.0, A 0, B 90, C 0} C_DIS
LIN {X -6.07, Y 59.68, Z 6.0, A 0, B 90, C 0} C_DIS
LIN {X -9.58, Y 59.23, Z 6.0, A 0, B 90, C 0} C_DIS
LIN {X -9.88, Y 59.17, Z 6.0, A 0, B 90, C 0} C_DIS
LIN {X -13.35, Y 58.5, Z 6.0, A 0, B 90, C 0} C_DIS
LIN {X -13.65, Y 58.42, Z 6.0, A 0, B 90, C 0} C_DIS
LIN {X -17.07, Y 57.52, Z 6.0, A 0, B 90, C 0} C_DIS
LIN {X -17.36, Y 57.42, Z 6.0, A 0, B 90, C 0} C_DIS
LIN {X -20.72, Y 56.31, Z 6.0, A 0, B 90, C 0} C_DIS
LIN {X -21.01, Y 56.19, Z 6.0, A 0, B 90, C 0} C_DIS
LIN {X -24.29, Y 54.86, Z 6.0, A 0, B 90, C 0} C_DIS
LIN {X -24.56, Y 54.73, Z 6.0, A 0, B 90, C 0} C_DIS
LIN {X -27.75, Y 53.2, Z 6.0, A 0, B 90, C 0} C_DIS
LIN {X -28.02, Y 53.04, Z 6.0, A 0, B 90, C 0} C_DIS
LIN {X -31.1, Y 51.31, Z 6.0, A 0, B 90, C 0} C_DIS
LIN {X -31.36, Y 51.14, Z 6.0, A 0, B 90, C 0} C_DIS
LIN {X -34.33, Y 49.21, Z 6.0, A 0, B 90, C 0} C_DIS
LIN {X -34.57, Y 49.03, Z 6.0, A 0, B 90, C 0} C_DIS
LIN {X -37.41, Y 46.91, Z 6.0, A 0, B 90, C 0} C_DIS
LIN {X -37.64, Y 46.71, Z 6.0, A 0, B 90, C 0} C_DIS
LIN {X -40.34, Y 44.42, Z 6.0, A 0, B 90, C 0} C_DIS
LIN {X -40.56, Y 44.2, Z 6.0, A 0, B 90, C 0} C_DIS
LIN {X -43.1, Y 41.74, Z 6.0, A 0, B 90, C 0} C_DIS
LIN {X -43.31, Y 41.51, Z 6.0, A 0, B 90, C 0} C_DIS
LIN {X -45.69, Y 38.89, Z 6.0, A 0, B 90, C 0} C_DIS
LIN {X -45.88, Y 38.65, Z 6.0, A 0, B 90, C 0} C_DIS
LIN {X -48.08, Y 35.89, Z 6.0, A 0, B 90, C 0} C_DIS
LIN {X -48.26, Y 35.63, Z 6.0, A 0, B 90, C 0} C_DIS
LIN {X -50.29, Y 32.73, Z 6.0, A 0, B 90, C 0} C_DIS
LIN {X -50.44, Y 32.47, Z 6.0, A 0, B 90, C 0} C_DIS
LIN {X -52.28, Y 29.44, Z 6.0, A 0, B 90, C 0} C_DIS
LIN {X -52.42, Y 29.17, Z 6.0, A 0, B 90, C 0} C_DIS
LIN {X -54.06, Y 26.03, Z 6.0, A 0, B 90, C 0} C_DIS
LIN {X -54.18, Y 25.75, Z 6.0, A 0, B 90, C 0} C_DIS
LIN {X -55.62, Y 22.52, Z 6.0, A 0, B 90, C 0} C_DIS
LIN {X -55.72, Y 22.23, Z 6.0, A 0, B 90, C 0} C_DIS
LIN {X -56.94, Y 18.91, Z 6.0, A 0, B 90, C 0} C_DIS
LIN {X -57.03, Y 18.61, Z 6.0, A 0, B 90, C 0} C_DIS
LIN {X -58.04, Y 15.22, Z 6.0, A 0, B 90, C 0} C_DIS
LIN {X -58.11, Y 14.92, Z 6.0, A 0, B 90, C 0} C_DIS
LIN {X -58.89, Y 11.47, Z 6.0, A 0, B 90, C 0} C_DIS
LIN {X -58.94, Y 11.17, Z 6.0, A 0, B 90, C 0} C_DIS
LIN {X -59.51, Y 7.67, Z 6.0, A 0, B 90, C 0} C_DIS
LIN {X -59.54, Y 7.37, Z 6.0, A 0, B 90, C 0} C_DIS
LIN {X -59.88, Y 3.84, Z 6.0, A 0, B 90, C 0} C_DIS
LIN {X -59.89, Y 3.54, Z 6.0, A 0, B 90, C 0} C_DIS
LIN {X -60.0, Y -0.0, Z 6.0, A 0, B 90, C 0} C_DIS
LIN {X -59.99, Y -0.31, Z 6.0, A 0, B 90, C 0} C_DIS
LIN {X -59.88, Y -3.84, Z 6.0, A 0, B 90, C 0} C_DIS
LIN {X -59.85, Y -4.15, Z 6.0, A 0, B 90, C 0} C_DIS
LIN {X -59.51, Y -7.67, Z 6.0, A 0, B 90, C 0} C_DIS
LIN {X -59.46, Y -7.98, Z 6.0, A 0, B 90, C 0} C_DIS
LIN {X -58.89, Y -11.47, Z 6.0, A 0, B 90, C 0} C_DIS
LIN {X -58.83, Y -11.77, Z 6.0, A 0, B 90, C 0} C_DIS
LIN {X -58.04, Y -15.22, Z 6.0, A 0, B 90, C 0} C_DIS
LIN {X -57.95, Y -15.51, Z 6.0, A 0, B 90, C 0} C_DIS
LIN {X -56.94, Y -18.91, Z 6.0, A 0, B 90, C 0} C_DIS
LIN {X -56.84, Y -19.2, Z 6.0, A 0, B 90, C 0} C_DIS
LIN {X -55.62, Y -22.52, Z 6.0, A 0, B 90, C 0} C_DIS
LIN {X -55.49, Y -22.8, Z 6.0, A 0, B 90, C 0} C_DIS
LIN {X -54.06, Y -26.03, Z 6.0, A 0, B 90, C 0} C_DIS
LIN {X -53.92, Y -26.31, Z 6.0, A 0, B 90, C 0} C_DIS
LIN {X -52.28, Y -29.44, Z 6.0, A 0, B 90, C 0} C_DIS
LIN {X -52.12, Y -29.71, Z 6.0, A 0, B 90, C 0} C_DIS
LIN {X -50.29, Y -32.73, Z 6.0, A 0, B 90, C 0} C_DIS
LIN {X -50.11, Y -32.98, Z 6.0, A 0, B 90, C 0} C_DIS
LIN {X -48.08, Y -35.89, Z 6.0, A 0, B 90, C 0} C_DIS
LIN {X -47.89, Y -36.13, Z 6.0, A 0, B 90, C 0} C_DIS
LIN {X -45.69, Y -38.89, Z 6.0, A 0, B 90, C 0} C_DIS
LIN {X -45.48, Y -39.12, Z 6.0, A 0, B 90, C 0} C_DIS
LIN {X -43.1, Y -41.74, Z 6.0, A 0, B 90, C 0} C_DIS
LIN {X -42.88, Y -41.96, Z 6.0, A 0, B 90, C 0} C_DIS
LIN {X -40.34, Y -44.42, Z 6.0, A 0, B 90, C 0} C_DIS
LIN {X -40.1, Y -44.62, Z 6.0, A 0, B 90, C 0} C_DIS
LIN {X -37.41, Y -46.91, Z 6.0, A 0, B 90, C 0} C_DIS
LIN {X -37.16, Y -47.09, Z 6.0, A 0, B 90, C 0} C_DIS
LIN {X -37.13, Y -47.11, Z 6.0, A 0, B 90, C 0} C_DIS
$OUT[1] = FALSE

; END LAYER 2
LIN {X -34.33, Y -49.21, Z 6.0, A 0, B 90, C 0} C_DIS
WAIT SEC 3
LIN {X -34.33, Y -49.21, Z 8.0, A 0, B 90, C 0} C_DIS
$OUT[1] = TRUE
WAIT SEC 0.8
LIN {X -34.33, Y -49.21, Z 8.0, A 0, B 90, C 0} C_DIS
LIN {X -34.33, Y -49.21, Z 8.0, A 0, B 90, C 0} C_DIS
LIN {X -33.94, Y -49.46, Z 8.0, A 0, B 90, C 0} C_DIS
LIN {X -31.1, Y -51.31, Z 8.0, A 0, B 90, C 0} C_DIS
LIN {X -30.7, Y -51.54, Z 8.0, A 0, B 90, C 0} C_DIS
LIN {X -27.75, Y -53.2, Z 8.0, A 0, B 90, C 0} C_DIS
LIN {X -27.34, Y -53.4, Z 8.0, A 0, B 90, C 0} C_DIS
LIN {X -24.29, Y -54.86, Z 8.0, A 0, B 90, C 0} C_DIS
LIN {X -23.86, Y -55.04, Z 8.0, A 0, B 90, C 0} C_DIS
LIN {X -20.72, Y -56.31, Z 8.0, A 0, B 90, C 0} C_DIS
LIN {X -20.28, Y -56.45, Z 8.0, A 0, B 90, C 0} C_DIS
LIN {X -17.07, Y -57.52, Z 8.0, A 0, B 90, C 0} C_DIS
LIN {X -16.63, Y -57.64, Z 8.0, A 0, B 90, C 0} C_DIS
LIN {X -13.35, Y -58.5, Z 8.0, A 0, B 90, C 0} C_DIS
LIN {X -12.9, Y -58.58, Z 8.0, A 0, B 90, C 0} C_DIS
LIN {X -9.58, Y -59.23, Z 8.0, A 0, B 90, C 0} C_DIS
LIN {X -9.12, Y -59.29, Z 8.0, A 0, B 90, C 0} C_DIS
LIN {X -5.76, Y -59.72, Z 8.0, A 0, B 90, C 0} C_DIS
LIN {X -5.3, Y -59.75, Z 8.0, A 0, B 90, C 0} C_DIS
LIN {X -1.92, Y -59.97, Z 8.0, A 0, B 90, C 0} C_DIS
LIN {X -1.46, Y -59.97, Z 8.0, A 0, B 90, C 0} C_DIS
LIN {X 1.92, Y -59.97, Z 8.0, A 0, B 90, C 0} C_DIS
LIN {X 2.38, Y -59.94, Z 8.0, A 0, B 90, C 0} C_DIS
LIN {X 5.76, Y -59.72, Z 8.0, A 0, B 90, C 0} C_DIS
LIN {X 6.22, Y -59.66, Z 8.0, A 0, B 90, C 0} C_DIS
LIN {X 9.58, Y -59.23, Z 8.0, A 0, B 90, C 0} C_DIS
LIN {X 10.03, Y -59.14, Z 8.0, A 0, B 90, C 0} C_DIS
LIN {X 13.35, Y -58.5, Z 8.0, A 0, B 90, C 0} C_DIS
LIN {X 13.8, Y -58.38, Z 8.0, A 0, B 90, C 0} C_DIS
LIN {X 17.07, Y -57.52, Z 8.0, A 0, B 90, C 0} C_DIS
LIN {X 17.51, Y -57.37, Z 8.0, A 0, B 90, C 0} C_DIS
LIN {X 20.72, Y -56.31, Z 8.0, A 0, B 90, C 0} C_DIS
LIN {X 21.15, Y -56.13, Z 8.0, A 0, B 90, C 0} C_DIS
LIN {X 24.29, Y -54.86, Z 8.0, A 0, B 90, C 0} C_DIS
LIN {X 24.7, Y -54.66, Z 8.0, A 0, B 90, C 0} C_DIS
LIN {X 27.75, Y -53.2, Z 8.0, A 0, B 90, C 0} C_DIS
LIN {X 28.15, Y -52.97, Z 8.0, A 0, B 90, C 0} C_DIS
LIN {X 31.1, Y -51.31, Z 8.0, A 0, B 90, C 0} C_DIS
LIN {X 31.49, Y -51.06, Z 8.0, A 0, B 90, C 0} C_DIS
LIN {X 34.33, Y -49.21, Z 8.0, A 0, B 90, C 0} C_DIS
LIN {X 34.7, Y -48.93, Z 8.0, A 0, B 90, C 0} C_DIS
LIN {X 37.41, Y -46.91, Z 8.0, A 0, B 90, C 0} C_DIS
LIN {X 37.76, Y -46.61, Z 8.0, A 0, B 90, C 0} C_DIS
LIN {X 40.34, Y -44.42, Z 8.0, A 0, B 90, C 0} C_DIS
LIN {X 40.67, Y -44.1, Z 8.0, A 0, B 90, C 0} C_DIS
LIN {X 43.1, Y -41.74, Z 8.0, A 0, B 90, C 0} C_DIS
LIN {X 43.41, Y -41.4, Z 8.0, A 0, B 90, C 0} C_DIS
LIN {X 45.69, Y -38.89, Z 8.0, A 0, B 90, C 0} C_DIS
LIN {X 45.97, Y -38.53, Z 8.0, A 0, B 90, C 0} C_DIS
LIN {X 48.08, Y -35.89, Z 8.0, A 0, B 90, C 0} C_DIS
LIN {X 48.35, Y -35.51, Z 8.0, A 0, B 90, C 0} C_DIS
LIN {X 50.29, Y -32.73, Z 8.0, A 0, B 90, C 0} C_DIS
LIN {X 50.52, Y -32.34, Z 8.0, A 0, B 90, C 0} C_DIS
LIN {X 52.28, Y -29.44, Z 8.0, A 0, B 90, C 0} C_DIS
LIN {X 52.49, Y -29.03, Z 8.0, A 0, B 90, C 0} C_DIS
LIN {X 54.06, Y -26.03, Z 8.0, A 0, B 90, C 0} C_DIS
LIN {X 54.24, Y -25.61, Z 8.0, A 0, B 90, C 0} C_DIS
LIN {X 55.62, Y -22.52, Z 8.0, A 0, B 90, C 0} C_DIS
LIN {X 55.77, Y -22.08, Z 8.0, A 0, B 90, C 0} C_DIS
LIN {X 56.94, Y -18.91, Z 8.0, A 0, B 90, C 0} C_DIS
LIN {X 57.07, Y -18.46, Z 8.0, A 0, B 90, C 0} C_DIS
LIN {X 58.04, Y -15.22, Z 8.0, A 0, B 90, C 0} C_DIS
LIN {X 58.14, Y -14.77, Z 8.0, A 0, B 90, C 0} C_DIS
LIN {X 58.89, Y -11.47, Z 8.0, A 0, B 90, C 0} C_DIS
LIN {X 58.97, Y -11.01, Z 8.0, A 0, B 90, C 0} C_DIS
LIN {X 59.51, Y -7.67, Z 8.0, A 0, B 90, C 0} C_DIS
LIN {X 59.55, Y -7.21, Z 8.0, A 0, B 90, C 0} C_DIS
LIN {X 59.88, Y -3.84, Z 8.0, A 0, B 90, C 0} C_DIS
LIN {X 59.89, Y -3.38, Z 8.0, A 0, B 90, C 0} C_DIS
LIN {X 60.0, Y 0.0, Z 8.0, A 0, B 90, C 0} C_DIS
LIN {X 59.99, Y 0.46, Z 8.0, A 0, B 90, C 0} C_DIS
LIN {X 59.88, Y 3.84, Z 8.0, A 0, B 90, C 0} C_DIS
LIN {X 59.83, Y 4.3, Z 8.0, A 0, B 90, C 0} C_DIS
LIN {X 59.51, Y 7.67, Z 8.0, A 0, B 90, C 0} C_DIS
LIN {X 59.43, Y 8.13, Z 8.0, A 0, B 90, C 0} C_DIS
LIN {X 58.89, Y 11.47, Z 8.0, A 0, B 90, C 0} C_DIS
LIN {X 58.79, Y 11.92, Z 8.0, A 0, B 90, C 0} C_DIS
LIN {X 58.04, Y 15.22, Z 8.0, A 0, B 90, C 0} C_DIS
LIN {X 57.91, Y 15.66, Z 8.0, A 0, B 90, C 0} C_DIS
LIN {X 56.94, Y 18.91, Z 8.0, A 0, B 90, C 0} C_DIS
LIN {X 56.78, Y 19.34, Z 8.0, A 0, B 90, C 0} C_DIS
LIN {X 55.62, Y 22.52, Z 8.0, A 0, B 90, C 0} C_DIS
LIN {X 55.43, Y 22.94, Z 8.0, A 0, B 90, C 0} C_DIS
LIN {X 54.06, Y 26.03, Z 8.0, A 0, B 90, C 0} C_DIS
LIN {X 53.84, Y 26.44, Z 8.0, A 0, B 90, C 0} C_DIS
LIN {X 52.28, Y 29.44, Z 8.0, A 0, B 90, C 0} C_DIS
LIN {X 52.04, Y 29.84, Z 8.0, A 0, B 90, C 0} C_DIS
LIN {X 50.29, Y 32.73, Z 8.0, A 0, B 90, C 0} C_DIS
LIN {X 50.02, Y 33.11, Z 8.0, A 0, B 90, C 0} C_DIS
LIN {X 48.08, Y 35.89, Z 8.0, A 0, B 90, C 0} C_DIS
LIN {X 47.8, Y 36.25, Z 8.0, A 0, B 90, C 0} C_DIS
LIN {X 45.69, Y 38.89, Z 8.0, A 0, B 90, C 0} C_DIS
LIN {X 45.38, Y 39.24, Z 8.0, A 0, B 90, C 0} C_DIS
LIN {X 43.1, Y 41.74, Z 8.0, A 0, B 90, C 0} C_DIS
LIN {X 42.77, Y 42.06, Z 8.0, A 0, B 90, C 0} C_DIS
LIN {X 40.34, Y 44.42, Z 8.0, A 0, B 90, C 0} C_DIS
LIN {X 39.99, Y 44.72, Z 8.0, A 0, B 90, C 0} C_DIS
LIN {X 37.41, Y 46.91, Z 8.0, A 0, B 90, C 0} C_DIS
LIN {X 37.04, Y 47.19, Z 8.0, A 0, B 90, C 0} C_DIS
LIN {X 34.33, Y 49.21, Z 8.0, A 0, B 90, C 0} C_DIS
LIN {X 33.94, Y 49.46, Z 8.0, A 0, B 90, C 0} C_DIS
LIN {X 31.1, Y 51.31, Z 8.0, A 0, B 90, C 0} C_DIS
LIN {X 30.7, Y 51.54, Z 8.0, A 0, B 90, C 0} C_DIS
LIN {X 27.75, Y 53.2, Z 8.0, A 0, B 90, C 0} C_DIS
LIN {X 27.34, Y 53.4, Z 8.0, A 0, B 90, C 0} C_DIS
LIN {X 24.29, Y 54.86, Z 8.0, A 0, B 90, C 0} C_DIS
LIN {X 23.86, Y 55.04, Z 8.0, A 0, B 90, C 0} C_DIS
LIN {X 20.72, Y 56.31, Z 8.0, A 0, B 90, C 0} C_DIS
LIN {X 20.28, Y 56.45, Z 8.0, A 0, B 90, C 0} C_DIS
LIN {X 17.07, Y 57.52, Z 8.0, A 0, B 90, C 0} C_DIS
LIN {X 16.63, Y 57.64, Z 8.0, A 0, B 90, C 0} C_DIS
LIN {X 13.35, Y 58.5, Z 8.0, A 0, B 90, C 0} C_DIS
LIN {X 12.9, Y 58.58, Z 8.0, A 0, B 90, C 0} C_DIS
LIN {X 9.58, Y 59.23, Z 8.0, A 0, B 90, C 0} C_DIS
LIN {X 9.12, Y 59.29, Z 8.0, A 0, B 90, C 0} C_DIS
LIN {X 5.76, Y 59.72, Z 8.0, A 0, B 90, C 0} C_DIS
LIN {X 5.3, Y 59.75, Z 8.0, A 0, B 90, C 0} C_DIS
LIN {X 1.92, Y 59.97, Z 8.0, A 0, B 90, C 0} C_DIS
LIN {X 1.46, Y 59.97, Z 8.0, A 0, B 90, C 0} C_DIS
LIN {X -1.92, Y 59.97, Z 8.0, A 0, B 90, C 0} C_DIS
LIN {X -2.38, Y 59.94, Z 8.0, A 0, B 90, C 0} C_DIS
LIN {X -5.76, Y 59.72, Z 8.0, A 0, B 90, C 0} C_DIS
LIN {X -6.22, Y 59.66, Z 8.0, A 0, B 90, C 0} C_DIS
LIN {X -9.58, Y 59.23, Z 8.0, A 0, B 90, C 0} C_DIS
LIN {X -10.03, Y 59.14, Z 8.0, A 0, B 90, C 0} C_DIS
LIN {X -13.35, Y 58.5, Z 8.0, A 0, B 90, C 0} C_DIS
LIN {X -13.8, Y 58.38, Z 8.0, A 0, B 90, C 0} C_DIS
LIN {X -17.07, Y 57.52, Z 8.0, A 0, B 90, C 0} C_DIS
LIN {X -17.51, Y 57.37, Z 8.0, A 0, B 90, C 0} C_DIS
LIN {X -20.72, Y 56.31, Z 8.0, A 0, B 90, C 0} C_DIS
LIN {X -21.15, Y 56.13, Z 8.0, A 0, B 90, C 0} C_DIS
LIN {X -24.29, Y 54.86, Z 8.0, A 0, B 90, C 0} C_DIS
LIN {X -24.7, Y 54.66, Z 8.0, A 0, B 90, C 0} C_DIS
LIN {X -27.75, Y 53.2, Z 8.0, A 0, B 90, C 0} C_DIS
LIN {X -28.15, Y 52.97, Z 8.0, A 0, B 90, C 0} C_DIS
LIN {X -31.1, Y 51.31, Z 8.0, A 0, B 90, C 0} C_DIS
LIN {X -31.49, Y 51.06, Z 8.0, A 0, B 90, C 0} C_DIS
LIN {X -34.33, Y 49.21, Z 8.0, A 0, B 90, C 0} C_DIS
LIN {X -34.7, Y 48.93, Z 8.0, A 0, B 90, C 0} C_DIS
LIN {X -37.41, Y 46.91, Z 8.0, A 0, B 90, C 0} C_DIS
LIN {X -37.76, Y 46.61, Z 8.0, A 0, B 90, C 0} C_DIS
LIN {X -40.34, Y 44.42, Z 8.0, A 0, B 90, C 0} C_DIS
LIN {X -40.67, Y 44.1, Z 8.0, A 0, B 90, C 0} C_DIS
LIN {X -43.1, Y 41.74, Z 8.0, A 0, B 90, C 0} C_DIS
LIN {X -43.41, Y 41.4, Z 8.0, A 0, B 90, C 0} C_DIS
LIN {X -45.69, Y 38.89, Z 8.0, A 0, B 90, C 0} C_DIS
LIN {X -45.97, Y 38.53, Z 8.0, A 0, B 90, C 0} C_DIS
LIN {X -48.08, Y 35.89, Z 8.0, A 0, B 90, C 0} C_DIS
LIN {X -48.35, Y 35.51, Z 8.0, A 0, B 90, C 0} C_DIS
LIN {X -50.29, Y 32.73, Z 8.0, A 0, B 90, C 0} C_DIS
LIN {X -50.52, Y 32.34, Z 8.0, A 0, B 90, C 0} C_DIS
LIN {X -52.28, Y 29.44, Z 8.0, A 0, B 90, C 0} C_DIS
LIN {X -52.49, Y 29.03, Z 8.0, A 0, B 90, C 0} C_DIS
LIN {X -54.06, Y 26.03, Z 8.0, A 0, B 90, C 0} C_DIS
LIN {X -54.24, Y 25.61, Z 8.0, A 0, B 90, C 0} C_DIS
LIN {X -55.62, Y 22.52, Z 8.0, A 0, B 90, C 0} C_DIS
LIN {X -55.77, Y 22.08, Z 8.0, A 0, B 90, C 0} C_DIS
LIN {X -56.94, Y 18.91, Z 8.0, A 0, B 90, C 0} C_DIS
LIN {X -57.07, Y 18.46, Z 8.0, A 0, B 90, C 0} C_DIS
LIN {X -58.04, Y 15.22, Z 8.0, A 0, B 90, C 0} C_DIS
LIN {X -58.14, Y 14.77, Z 8.0, A 0, B 90, C 0} C_DIS
LIN {X -58.89, Y 11.47, Z 8.0, A 0, B 90, C 0} C_DIS
LIN {X -58.97, Y 11.01, Z 8.0, A 0, B 90, C 0} C_DIS
LIN {X -59.51, Y 7.67, Z 8.0, A 0, B 90, C 0} C_DIS
LIN {X -59.55, Y 7.21, Z 8.0, A 0, B 90, C 0} C_DIS
LIN {X -59.88, Y 3.84, Z 8.0, A 0, B 90, C 0} C_DIS
LIN {X -59.89, Y 3.38, Z 8.0, A 0, B 90, C 0} C_DIS
LIN {X -60.0, Y -0.0, Z 8.0, A 0, B 90, C 0} C_DIS
LIN {X -59.99, Y -0.46, Z 8.0, A 0, B 90, C 0} C_DIS
LIN {X -59.88, Y -3.84, Z 8.0, A 0, B 90, C 0} C_DIS
LIN {X -59.83, Y -4.3, Z 8.0, A 0, B 90, C 0} C_DIS
LIN {X -59.51, Y -7.67, Z 8.0, A 0, B 90, C 0} C_DIS
LIN {X -59.43, Y -8.13, Z 8.0, A 0, B 90, C 0} C_DIS
LIN {X -58.89, Y -11.47, Z 8.0, A 0, B 90, C 0} C_DIS
LIN {X -58.79, Y -11.92, Z 8.0, A 0, B 90, C 0} C_DIS
LIN {X -58.04, Y -15.22, Z 8.0, A 0, B 90, C 0} C_DIS
LIN {X -57.91, Y -15.66, Z 8.0, A 0, B 90, C 0} C_DIS
LIN {X -56.94, Y -18.91, Z 8.0, A 0, B 90, C 0} C_DIS
LIN {X -56.78, Y -19.34, Z 8.0, A 0, B 90, C 0} C_DIS
LIN {X -55.62, Y -22.52, Z 8.0, A 0, B 90, C 0} C_DIS
LIN {X -55.43, Y -22.94, Z 8.0, A 0, B 90, C 0} C_DIS
LIN {X -54.06, Y -26.03, Z 8.0, A 0, B 90, C 0} C_DIS
LIN {X -53.84, Y -26.44, Z 8.0, A 0, B 90, C 0} C_DIS
LIN {X -52.28, Y -29.44, Z 8.0, A 0, B 90, C 0} C_DIS
LIN {X -52.04, Y -29.84, Z 8.0, A 0, B 90, C 0} C_DIS
LIN {X -50.29, Y -32.73, Z 8.0, A 0, B 90, C 0} C_DIS
LIN {X -50.02, Y -33.11, Z 8.0, A 0, B 90, C 0} C_DIS
LIN {X -48.08, Y -35.89, Z 8.0, A 0, B 90, C 0} C_DIS
LIN {X -47.8, Y -36.25, Z 8.0, A 0, B 90, C 0} C_DIS
LIN {X -45.69, Y -38.89, Z 8.0, A 0, B 90, C 0} C_DIS
LIN {X -45.38, Y -39.24, Z 8.0, A 0, B 90, C 0} C_DIS
LIN {X -43.1, Y -41.74, Z 8.0, A 0, B 90, C 0} C_DIS
LIN {X -42.77, Y -42.06, Z 8.0, A 0, B 90, C 0} C_DIS
LIN {X -40.34, Y -44.42, Z 8.0, A 0, B 90, C 0} C_DIS
LIN {X -39.99, Y -44.72, Z 8.0, A 0, B 90, C 0} C_DIS
LIN {X -37.41, Y -46.91, Z 8.0, A 0, B 90, C 0} C_DIS
LIN {X -37.04, Y -47.19, Z 8.0, A 0, B 90, C 0} C_DIS
$OUT[1] = FALSE

; END LAYER 3
LIN {X -34.33, Y -49.21, Z 8.0, A 0, B 90, C 0} C_DIS
WAIT SEC 3
LIN {X -34.33, Y -49.21, Z 10.0, A 0, B 90, C 0} C_DIS
$OUT[1] = TRUE
WAIT SEC 0.8
LIN {X -34.33, Y -49.21, Z 10.0, A 0, B 90, C 0} C_DIS
LIN {X -34.33, Y -49.21, Z 10.0, A 0, B 90, C 0} C_DIS
LIN {X -33.81, Y -49.55, Z 10.0, A 0, B 90, C 0} C_DIS
LIN {X -31.1, Y -51.31, Z 10.0, A 0, B 90, C 0} C_DIS
LIN {X -30.57, Y -51.61, Z 10.0, A 0, B 90, C 0} C_DIS
LIN {X -27.75, Y -53.2, Z 10.0, A 0, B 90, C 0} C_DIS
LIN {X -27.2, Y -53.46, Z 10.0, A 0, B 90, C 0} C_DIS
LIN {X -24.29, Y -54.86, Z 10.0, A 0, B 90, C 0} C_DIS
LIN {X -23.72, Y -55.1, Z 10.0, A 0, B 90, C 0} C_DIS
LIN {X -20.72, Y -56.31, Z 10.0, A 0, B 90, C 0} C_DIS
LIN {X -20.14, Y -56.5, Z 10.0, A 0, B 90, C 0} C_DIS
LIN {X -17.07, Y -57.52, Z 10.0, A 0, B 90, C 0} C_DIS
LIN {X -16.48, Y -57.68, Z 10.0, A 0, B 90, C 0} C_DIS
LIN {X -13.35, Y -58.5, Z 10.0, A 0, B 90, C 0} C_DIS
LIN {X -12.75, Y -58.61, Z 10.0, A 0, B 90, C 0} C_DIS
LIN {X -9.58, Y -59.23, Z 10.0, A 0, B 90, C 0} C_DIS
LIN {X -8.97, Y -59.31, Z 10.0, A 0, B 90, C 0} C_DIS
LIN {X -5.76, Y -59.72, Z 10.0, A 0, B 90, C 0} C_DIS
LIN {X -5.15, Y -59.76, Z 10.0, A 0, B 90, C 0} C_DIS
LIN {X -1.92, Y -59.97, Z 10.0, A 0, B 90, C 0} C_DIS
LIN {X -1.31, Y -59.97, Z 10.0, A 0, B 90, C 0} C_DIS
LIN {X 1.92, Y -59.97, Z 10.0, A 0, B 90, C 0} C_DIS
LIN {X 2.54, Y -59.93, Z 10.0, A 0, B 90, C 0} C_DIS
LIN {X 5.76, Y -59.72, Z 10.0, A 0, B 90, C 0} C_DIS
LIN {X 6.37, Y -59.64, Z 10.0, A 0, B 90, C 0} C_DIS
LIN {X 9.58, Y -59.23, Z 10.0, A 0, B 90, C 0} C_DIS
LIN {X 10.18, Y -59.11, Z 10.0, A 0, B 90, C 0} C_DIS
LIN {X 13.35, Y -58.5, Z 10.0, A 0, B 90, C 0} C_DIS
LIN {X 13.95, Y -58.34, Z 10.0, A 0, B 90, C 0} C_DIS
LIN {X 17.07, Y -57.52, Z 10.0, A 0, B 90, C 0} C_DIS
LIN {X 17.66, Y -57.33, Z 10.0, A 0, B 90, C 0} C_DIS
LIN {X 20.72, Y -56.31, Z 10.0, A 0, B 90, C 0} C_DIS
LIN {X 21.29, Y -56.08, Z 10.0, A 0, B 90, C 0} C_DIS
LIN {X 24.29, Y -54.86, Z 10.0, A 0, B 90, C 0} C_DIS
LIN {X 24.84, Y -54.6, Z 10.0, A 0, B 90, C 0} C_DIS
LIN {X 27.75, Y -53.2, Z 10.0, A 0, B 90, C 0} C_DIS
LIN {X 28.29, Y -52.89, Z 10.0, A 0, B 90, C 0} C_DIS
LIN {X 31.1, Y -51.31, Z 10.0, A 0, B 90, C 0} C_DIS
LIN {X 31.62, Y -50.97, Z 10.0, A 0, B 90, C 0} C_DIS
LIN {X 34.33, Y -49.21, Z 10.0, A 0, B 90, C 0} C_DIS
LIN {X 34.82, Y -48.84, Z 10.0, A 0, B 90, C 0} C_DIS
LIN {X 37.41, Y -46.91, Z 10.0, A 0, B 90, C 0} C_DIS
LIN {X 37.88, Y -46.51, Z 10.0, A 0, B 90, C 0} C_DIS
LIN {X 40.34, Y -44.42, Z 10.0, A 0, B 90, C 0} C_DIS
LIN {X 40.78, Y -43.99, Z 10.0, A 0, B 90, C 0} C_DIS
LIN {X 43.1, Y -41.74, Z 10.0, A 0, B 90, C 0} C_DIS
LIN {X 43.51, Y -41.29, Z 10.0, A 0, B 90, C 0} C_DIS
LIN {X 45.69, Y -38.89, Z 10.0, A 0, B 90, C 0} C_DIS
LIN {X 46.07, Y -38.41, Z 10.0, A 0, B 90, C 0} C_DIS
LIN {X 48.08, Y -35.89, Z 10.0, A 0, B 90, C 0} C_DIS
LIN {X 48.44, Y -35.38, Z 10.0, A 0, B 90, C 0} C_DIS
LIN {X 50.29, Y -32.73, Z 10.0, A 0, B 90, C 0} C_DIS
LIN {X 50.6, Y -32.21, Z 10.0, A 0, B 90, C 0} C_DIS
LIN {X 52.28, Y -29.44, Z 10.0, A 0, B 90, C 0} C_DIS
LIN {X 52.56, Y -28.9, Z 10.0, A 0, B 90, C 0} C_DIS
LIN {X 54.06, Y -26.03, Z 10.0, A 0, B 90, C 0} C_DIS
LIN {X 54.31, Y -25.47, Z 10.0, A 0, B 90, C 0} C_DIS
LIN {X 55.62, Y -22.52, Z 10.0, A 0, B 90, C 0} C_DIS
LIN {X 55.83, Y -21.94, Z 10.0, A 0, B 90, C 0} C_DIS
LIN {X 56.94, Y -18.91, Z 10.0, A 0, B 90, C 0} C_DIS
LIN {X 57.12, Y -18.32, Z 10.0, A 0, B 90, C 0} C_DIS
LIN {X 58.04, Y -15.22, Z 10.0, A 0, B 90, C 0} C_DIS
LIN {X 58.17, Y -14.62, Z 10.0, A 0, B 90, C 0} C_DIS
LIN {X 58.89, Y -11.47, Z 10.0, A 0, B 90, C 0} C_DIS
LIN {X 58.99, Y -10.86, Z 10.0, A 0, B 90, C 0} C_DIS
LIN {X 59.51, Y -7.67, Z 10.0, A 0, B 90, C 0} C_DIS
LIN {X 59.57, Y -7.06, Z 10.0, A 0, B 90, C 0} C_DIS
LIN {X 59.88, Y -3.84, Z 10.0, A 0, B 90, C 0} C_DIS
LIN {X 59.9, Y -3.23, Z 10.0, A 0, B 90, C 0} C_DIS
LIN {X 60.0, Y 0.0, Z 10.0, A 0, B 90, C 0} C_DIS
LIN {X 59.98, Y 0.62, Z 10.0, A 0, B 90, C 0} C_DIS
LIN {X 59.88, Y 3.84, Z 10.0, A 0, B 90, C 0} C_DIS
LIN {X 59.82, Y 4.46, Z 10.0, A 0, B 90, C 0} C_DIS
LIN {X 59.51, Y 7.67, Z 10.0, A 0, B 90, C 0} C_DIS
LIN {X 59.41, Y 8.28, Z 10.0, A 0, B 90, C 0} C_DIS
LIN {X 58.89, Y 11.47, Z 10.0, A 0, B 90, C 0} C_DIS
LIN {X 58.76, Y 12.07, Z 10.0, A 0, B 90, C 0} C_DIS
LIN {X 58.04, Y 15.22, Z 10.0, A 0, B 90, C 0} C_DIS
LIN {X 57.86, Y 15.81, Z 10.0, A 0, B 90, C 0} C_DIS
LIN {X 56.94, Y 18.91, Z 10.0, A 0, B 90, C 0} C_DIS
LIN {X 56.73, Y 19.48, Z 10.0, A 0, B 90, C 0} C_DIS
LIN {X 55.62, Y 22.52, Z 10.0, A 0, B 90, C 0} C_DIS
LIN {X 55.37, Y 23.08, Z 10.0, A 0, B 90, C 0} C_DIS
LIN {X 54.06, Y 26.03, Z 10.0, A 0, B 90, C 0} C_DIS
LIN {X 53.77, Y 26.58, Z 10.0, A 0, B 90, C 0} C_DIS
LIN {X 52.28, Y 29.44, Z 10.0, A 0, B 90, C 0} C_DIS
LIN {X 51.96, Y 29.97, Z 10.0, A 0, B 90, C 0} C_DIS
LIN {X 50.29, Y 32.73, Z 10.0, A 0, B 90, C 0} C_DIS
LIN {X 49.93, Y 33.24, Z 10.0, A 0, B 90, C 0} C_DIS
LIN {X 48.08, Y 35.89, Z 10.0, A 0, B 90, C 0} C_DIS
LIN {X 47.7, Y 36.37, Z 10.0, A 0, B 90, C 0} C_DIS
LIN {X 45.69, Y 38.89, Z 10.0, A 0, B 90, C 0} C_DIS
LIN {X 45.27, Y 39.35, Z 10.0, A 0, B 90, C 0} C_DIS
LIN {X 43.1, Y 41.74, Z 10.0, A 0, B 90, C 0} C_DIS
LIN {X 42.66, Y 42.17, Z 10.0, A 0, B 90, C 0} C_DIS
LIN {X 40.34, Y 44.42, Z 10.0, A 0, B 90, C 0} C_DIS
LIN {X 39.87, Y 44.82, Z 10.0, A 0, B 90, C 0} C_DIS
LIN {X 37.41, Y 46.91, Z 10.0, A 0, B 90, C 0} C_DIS
LIN {X 36.92, Y 47.28, Z 10.0, A 0, B 90, C 0} C_DIS
LIN {X 34.33, Y 49.21, Z 10.0, A 0, B 90, C 0} C_DIS
LIN {X 33.81, Y 49.55, Z 10.0, A 0, B 90, C 0} C_DIS
LIN {X 31.1, Y 51.31, Z 10.0, A 0, B 90, C 0} C_DIS
LIN {X 30.57, Y 51.61, Z 10.0, A 0, B 90, C 0} C_DIS
LIN {X 27.75, Y 53.2, Z 10.0, A 0, B 90, C 0} C_DIS
LIN {X 27.2, Y 53.46, Z 10.0, A 0, B 90, C 0} C_DIS
LIN {X 24.29, Y 54.86, Z 10.0, A 0, B 90, C 0} C_DIS
LIN {X 23.72, Y 55.1, Z 10.0, A 0, B 90, C 0} C_DIS
LIN {X 20.72, Y 56.31, Z 10.0, A 0, B 90, C 0} C_DIS
LIN {X 20.14, Y 56.5, Z 10.0, A 0, B 90, C 0} C_DIS
LIN {X 17.07, Y 57.52, Z 10.0, A 0, B 90, C 0} C_DIS
LIN {X 16.48, Y 57.68, Z 10.0, A 0, B 90, C 0} C_DIS
LIN {X 13.35, Y 58.5, Z 10.0, A 0, B 90, C 0} C_DIS
LIN {X 12.75, Y 58.61, Z 10.0, A 0, B 90, C 0} C_DIS
LIN {X 9.58, Y 59.23, Z 10.0, A 0, B 90, C 0} C_DIS
LIN {X 8.97, Y 59.31, Z 10.0, A 0, B 90, C 0} C_DIS
LIN {X 5.76, Y 59.72, Z 10.0, A 0, B 90, C 0} C_DIS
LIN {X 5.15, Y 59.76, Z 10.0, A 0, B 90, C 0} C_DIS
LIN {X 1.92, Y 59.97, Z 10.0, A 0, B 90, C 0} C_DIS
LIN {X 1.31, Y 59.97, Z 10.0, A 0, B 90, C 0} C_DIS
LIN {X -1.92, Y 59.97, Z 10.0, A 0, B 90, C 0} C_DIS
LIN {X -2.54, Y 59.93, Z 10.0, A 0, B 90, C 0} C_DIS
LIN {X -5.76, Y 59.72, Z 10.0, A 0, B 90, C 0} C_DIS
LIN {X -6.37, Y 59.64, Z 10.0, A 0, B 90, C 0} C_DIS
LIN {X -9.58, Y 59.23, Z 10.0, A 0, B 90, C 0} C_DIS
LIN {X -10.18, Y 59.11, Z 10.0, A 0, B 90, C 0} C_DIS
LIN {X -13.35, Y 58.5, Z 10.0, A 0, B 90, C 0} C_DIS
LIN {X -13.95, Y 58.34, Z 10.0, A 0, B 90, C 0} C_DIS
LIN {X -17.07, Y 57.52, Z 10.0, A 0, B 90, C 0} C_DIS
LIN {X -17.66, Y 57.33, Z 10.0, A 0, B 90, C 0} C_DIS
LIN {X -20.72, Y 56.31, Z 10.0, A 0, B 90, C 0} C_DIS
LIN {X -21.29, Y 56.08, Z 10.0, A 0, B 90, C 0} C_DIS
LIN {X -24.29, Y 54.86, Z 10.0, A 0, B 90, C 0} C_DIS
LIN {X -24.84, Y 54.6, Z 10.0, A 0, B 90, C 0} C_DIS
LIN {X -27.75, Y 53.2, Z 10.0, A 0, B 90, C 0} C_DIS
LIN {X -28.29, Y 52.89, Z 10.0, A 0, B 90, C 0} C_DIS
LIN {X -31.1, Y 51.31, Z 10.0, A 0, B 90, C 0} C_DIS
LIN {X -31.62, Y 50.97, Z 10.0, A 0, B 90, C 0} C_DIS
LIN {X -34.33, Y 49.21, Z 10.0, A 0, B 90, C 0} C_DIS
LIN {X -34.82, Y 48.84, Z 10.0, A 0, B 90, C 0} C_DIS
LIN {X -37.41, Y 46.91, Z 10.0, A 0, B 90, C 0} C_DIS
LIN {X -37.88, Y 46.51, Z 10.0, A 0, B 90, C 0} C_DIS
LIN {X -40.34, Y 44.42, Z 10.0, A 0, B 90, C 0} C_DIS
LIN {X -40.78, Y 43.99, Z 10.0, A 0, B 90, C 0} C_DIS
LIN {X -43.1, Y 41.74, Z 10.0, A 0, B 90, C 0} C_DIS
LIN {X -43.51, Y 41.29, Z 10.0, A 0, B 90, C 0} C_DIS
LIN {X -45.69, Y 38.89, Z 10.0, A 0, B 90, C 0} C_DIS
LIN {X -46.07, Y 38.41, Z 10.0, A 0, B 90, C 0} C_DIS
LIN {X -48.08, Y 35.89, Z 10.0, A 0, B 90, C 0} C_DIS
LIN {X -48.44, Y 35.38, Z 10.0, A 0, B 90, C 0} C_DIS
LIN {X -50.29, Y 32.73, Z 10.0, A 0, B 90, C 0} C_DIS
LIN {X -50.6, Y 32.21, Z 10.0, A 0, B 90, C 0} C_DIS
LIN {X -52.28, Y 29.44, Z 10.0, A 0, B 90, C 0} C_DIS
LIN {X -52.56, Y 28.9, Z 10.0, A 0, B 90, C 0} C_DIS
LIN {X -54.06, Y 26.03, Z 10.0, A 0, B 90, C 0} C_DIS
LIN {X -54.31, Y 25.47, Z 10.0, A 0, B 90, C 0} C_DIS
LIN {X -55.62, Y 22.52, Z 10.0, A 0, B 90, C 0} C_DIS
LIN {X -55.83, Y 21.94, Z 10.0, A 0, B 90, C 0} C_DIS
LIN {X -56.94, Y 18.91, Z 10.0, A 0, B 90, C 0} C_DIS
LIN {X -57.12, Y 18.32, Z 10.0, A 0, B 90, C 0} C_DIS
LIN {X -58.04, Y 15.22, Z 10.0, A 0, B 90, C 0} C_DIS
LIN {X -58.17, Y 14.62, Z 10.0, A 0, B 90, C 0} C_DIS
LIN {X -58.89, Y 11.47, Z 10.0, A 0, B 90, C 0} C_DIS
LIN {X -58.99, Y 10.86, Z 10.0, A 0, B 90, C 0} C_DIS
LIN {X -59.51, Y 7.67, Z 10.0, A 0, B 90, C 0} C_DIS
LIN {X -59.57, Y 7.06, Z 10.0, A 0, B 90, C 0} C_DIS
LIN {X -59.88, Y 3.84, Z 10.0, A 0, B 90, C 0} C_DIS
LIN {X -59.9, Y 3.23, Z 10.0, A 0, B 90, C 0} C_DIS
LIN {X -60.0, Y -0.0, Z 10.0, A 0, B 90, C 0} C_DIS
LIN {X -59.98, Y -0.62, Z 10.0, A 0, B 90, C 0} C_DIS
LIN {X -59.88, Y -3.84, Z 10.0, A 0, B 90, C 0} C_DIS
LIN {X -59.82, Y -4.46, Z 10.0, A 0, B 90, C 0} C_DIS
LIN {X -59.51, Y -7.67, Z 10.0, A 0, B 90, C 0} C_DIS
LIN {X -59.41, Y -8.28, Z 10.0, A 0, B 90, C 0} C_DIS
LIN {X -58.89, Y -11.47, Z 10.0, A 0, B 90, C 0} C_DIS
LIN {X -58.76, Y -12.07, Z 10.0, A 0, B 90, C 0} C_DIS
LIN {X -58.04, Y -15.22, Z 10.0, A 0, B 90, C 0} C_DIS
LIN {X -57.86, Y -15.81, Z 10.0, A 0, B 90, C 0} C_DIS
LIN {X -56.94, Y -18.91, Z 10.0, A 0, B 90, C 0} C_DIS
LIN {X -56.73, Y -19.48, Z 10.0, A 0, B 90, C 0} C_DIS
LIN {X -55.62, Y -22.52, Z 10.0, A 0, B 90, C 0} C_DIS
LIN {X -55.37, Y -23.08, Z 10.0, A 0, B 90, C 0} C_DIS
LIN {X -54.06, Y -26.03, Z 10.0, A 0, B 90, C 0} C_DIS
LIN {X -53.77, Y -26.58, Z 10.0, A 0, B 90, C 0} C_DIS
LIN {X -52.28, Y -29.44, Z 10.0, A 0, B 90, C 0} C_DIS
LIN {X -51.96, Y -29.97, Z 10.0, A 0, B 90, C 0} C_DIS
LIN {X -50.29, Y -32.73, Z 10.0, A 0, B 90, C 0} C_DIS
LIN {X -49.93, Y -33.24, Z 10.0, A 0, B 90, C 0} C_DIS
LIN {X -48.08, Y -35.89, Z 10.0, A 0, B 90, C 0} C_DIS
LIN {X -47.7, Y -36.37, Z 10.0, A 0, B 90, C 0} C_DIS
LIN {X -45.69, Y -38.89, Z 10.0, A 0, B 90, C 0} C_DIS
LIN {X -45.27, Y -39.35, Z 10.0, A 0, B 90, C 0} C_DIS
LIN {X -43.1, Y -41.74, Z 10.0, A 0, B 90, C 0} C_DIS
LIN {X -42.66, Y -42.17, Z 10.0, A 0, B 90, C 0} C_DIS
LIN {X -40.34, Y -44.42, Z 10.0, A 0, B 90, C 0} C_DIS
LIN {X -39.87, Y -44.82, Z 10.0, A 0, B 90, C 0} C_DIS
LIN {X -37.41, Y -46.91, Z 10.0, A 0, B 90, C 0} C_DIS
LIN {X -36.92, Y -47.28, Z 10.0, A 0, B 90, C 0} C_DIS
$OUT[1] = FALSE

; END LAYER 4
LIN {X -34.33, Y -49.21, Z 10.0, A 0, B 90, C 0} C_DIS
WAIT SEC 3
LIN {X -34.33, Y -49.21, Z 12.0, A 0, B 90, C 0} C_DIS
$OUT[1] = TRUE
WAIT SEC 0.8
LIN {X -34.33, Y -49.21, Z 12.0, A 0, B 90, C 0} C_DIS
LIN {X -34.33, Y -49.21, Z 12.0, A 0, B 90, C 0} C_DIS
LIN {X -33.68, Y -49.63, Z 12.0, A 0, B 90, C 0} C_DIS
LIN {X -31.1, Y -51.31, Z 12.0, A 0, B 90, C 0} C_DIS
LIN {X -30.43, Y -51.69, Z 12.0, A 0, B 90, C 0} C_DIS
LIN {X -27.75, Y -53.2, Z 12.0, A 0, B 90, C 0} C_DIS
LIN {X -27.06, Y -53.53, Z 12.0, A 0, B 90, C 0} C_DIS
LIN {X -24.29, Y -54.86, Z 12.0, A 0, B 90, C 0} C_DIS
LIN {X -23.57, Y -55.15, Z 12.0, A 0, B 90, C 0} C_DIS
LIN {X -20.72, Y -56.31, Z 12.0, A 0, B 90, C 0} C_DIS
LIN {X -19.99, Y -56.55, Z 12.0, A 0, B 90, C 0} C_DIS
LIN {X -17.07, Y -57.52, Z 12.0, A 0, B 90, C 0} C_DIS
LIN {X -16.33, Y -57.72, Z 12.0, A 0, B 90, C 0} C_DIS
LIN {X -13.35, Y -58.5, Z 12.0, A 0, B 90, C 0} C_DIS
LIN {X -12.6, Y -58.64, Z 12.0, A 0, B 90, C 0} C_DIS
LIN {X -9.58, Y -59.23, Z 12.0, A 0, B 90, C 0} C_DIS
LIN {X -8.81, Y -59.33, Z 12.0, A 0, B 90, C 0} C_DIS
LIN {X -5.76, Y -59.72, Z 12.0, A 0, B 90, C 0} C_DIS
LIN {X -4.99, Y -59.77, Z 12.0, A 0, B 90, C 0} C_DIS
LIN {X -1.92, Y -59.97, Z 12.0, A 0, B 90, C 0} C_DIS
LIN {X -1.15, Y -59.97, Z 12.0, A 0, B 90, C 0} C_DIS
LIN {X 1.92, Y -59.97, Z 12.0, A 0, B 90, C 0} C_DIS
LIN {X 2.69, Y -59.92, Z 12.0, A 0, B 90, C 0} C_DIS
LIN {X 5.76, Y -59.72, Z 12.0, A 0, B 90, C 0} C_DIS
LIN {X 6.52, Y -59.62, Z 12.0, A 0, B 90, C 0} C_DIS
LIN {X 9.58, Y -59.23, Z 12.0, A 0, B 90, C 0} C_DIS
LIN {X 10.33, Y -59.08, Z 12.0, A 0, B 90, C 0} C_DIS
LIN {X 13.35, Y -58.5, Z 12.0, A 0, B 90, C 0} C_DIS
LIN {X 14.1, Y -58.3, Z 12.0, A 0, B 90, C 0} C_DIS
LIN {X 17.07, Y -57.52, Z 12.0, A 0, B 90, C 0} C_DIS
LIN {X 17.8, Y -57.28, Z 12.0, A 0, B 90, C 0} C_DIS
LIN {X 20.72, Y -56.31, Z 12.0, A 0, B 90, C 0} C_DIS
LIN {X 21.43, Y -56.02, Z 12.0, A 0, B 90, C 0} C_DIS
LIN {X 24.29, Y -54.86, Z 12.0, A 0, B 90, C 0} C_DIS
LIN {X 24.98, Y -54.53, Z 12.0, A 0, B 90, C 0} C_DIS
LIN {X 27.75, Y -53.2, Z 12.0, A 0, B 90, C 0} C_DIS
LIN {X 28.42, Y -52.82, Z 12.0, A 0, B 90, C 0} C_DIS
LIN {X 31.1, Y -51.31, Z 12.0, A 0, B 90, C 0} C_DIS
LIN {X 31.75, Y -50.89, Z 12.0, A 0, B 90, C 0} C_DIS
LIN {X 34.33, Y -49.21, Z 12.0, A 0, B 90, C 0} C_DIS
LIN {X 34.94, Y -48.75, Z 12.0, A 0, B 90, C 0} C_DIS
LIN {X 37.41, Y -46.91, Z 12.0, A 0, B 90, C 0} C_DIS
LIN {X 38.0, Y -46.41, Z 12.0, A 0, B 90, C 0} C_DIS
LIN {X 40.34, Y -44.42, Z 12.0, A 0, B 90, C 0} C_DIS
LIN {X 40.89, Y -43.88, Z 12.0, A 0, B 90, C 0} C_DIS
LIN {X 43.1, Y -41.74, Z 12.0, A 0, B 90, C 0} C_DIS
LIN {X 43.62, Y -41.17, Z 12.0, A 0, B 90, C 0} C_DIS
LIN {X 45.69, Y -38.89, Z 12.0, A 0, B 90, C 0} C_DIS
LIN {X 46.17, Y -38.29, Z 12.0, A 0, B 90, C 0} C_DIS
LIN {X 48.08, Y -35.89, Z 12.0, A 0, B 90, C 0} C_DIS
LIN {X 48.52, Y -35.26, Z 12.0, A 0, B 90, C 0} C_DIS
LIN {X 50.29, Y -32.73, Z 12.0, A 0, B 90, C 0} C_DIS
LIN {X 50.68, Y -32.07, Z 12.0, A 0, B 90, C 0} C_DIS
LIN {X 52.28, Y -29.44, Z 12.0, A 0, B 90, C 0} C_DIS
LIN {X 52.63, Y -28.76, Z 12.0, A 0, B 90, C 0} C_DIS
LIN {X 54.06, Y -26.03, Z 12.0, A 0, B 90, C 0} C_DIS
LIN {X 54.37, Y -25.33, Z 12.0, A 0, B 90, C 0} C_DIS
LIN {X 55.62, Y -22.52, Z 12.0, A 0, B 90, C 0} C_DIS
LIN {X 55.88, Y -21.79, Z 12.0, A 0, B 90, C 0} C_DIS
LIN {X 56.94, Y -18.91, Z 12.0, A 0, B 90, C 0} C_DIS
LIN {X 57.16, Y -18.17, Z 12.0, A 0, B 90, C 0} C_DIS
LIN {X 58.04, Y -15.22, Z 12.0, A 0, B 90, C 0} C_DIS
LIN {X 58.21, Y -14.47, Z 12.0, A 0, B 90, C 0} C_DIS
LIN {X 58.89, Y -11.47, Z 12.0, A 0, B 90, C 0} C_DIS
LIN {X 59.02, Y -10.71, Z 12.0, A 0, B 90, C 0} C_DIS
LIN {X 59.51, Y -7.67, Z 12.0, A 0, B 90, C 0} C_DIS
LIN {X 59.58, Y -6.91, Z 12.0, A 0, B 90, C 0} C_DIS
LIN {X 59.88, Y -3.84, Z 12.0, A 0, B 90, C 0} C_DIS
LIN {X 59.9, Y -3.08, Z 12.0, A 0, B 90, C 0} C_DIS
LIN {X 60.0, Y -0.0, Z 12.0, A 0, B 90, C 0} C_DIS
LIN {X 59.98, Y 0.77, Z 12.0, A 0, B 90, C 0} C_DIS
LIN {X 59.88, Y 3.84, Z 12.0, A 0, B 90, C 0} C_DIS
LIN {X 59.8, Y 4.61, Z 12.0, A 0, B 90, C 0} C_DIS
LIN {X 59.51, Y 7.67, Z 12.0, A 0, B 90, C 0} C_DIS
LIN {X 59.38, Y 8.43, Z 12.0, A 0, B 90, C 0} C_DIS
LIN {X 58.89, Y 11.47, Z 12.0, A 0, B 90, C 0} C_DIS
LIN {X 58.72, Y 12.22, Z 12.0, A 0, B 90, C 0} C_DIS
LIN {X 58.04, Y 15.22, Z 12.0, A 0, B 90, C 0} C_DIS
LIN {X 57.82, Y 15.96, Z 12.0, A 0, B 90, C 0} C_DIS
LIN {X 56.94, Y 18.91, Z 12.0, A 0, B 90, C 0} C_DIS
LIN {X 56.68, Y 19.63, Z 12.0, A 0, B 90, C 0} C_DIS
LIN {X 55.62, Y 22.52, Z 12.0, A 0, B 90, C 0} C_DIS
LIN {X 55.3, Y 23.22, Z 12.0, A 0, B 90, C 0} C_DIS
LIN {X 54.06, Y 26.03, Z 12.0, A 0, B 90, C 0} C_DIS
LIN {X 53.7, Y 26.72, Z 12.0, A 0, B 90, C 0} C_DIS
LIN {X 52.28, Y 29.44, Z 12.0, A 0, B 90, C 0} C_DIS
LIN {X 51.88, Y 30.1, Z 12.0, A 0, B 90, C 0} C_DIS
LIN {X 50.29, Y 32.73, Z 12.0, A 0, B 90, C 0} C_DIS
LIN {X 49.85, Y 33.36, Z 12.0, A 0, B 90, C 0} C_DIS
LIN {X 48.08, Y 35.89, Z 12.0, A 0, B 90, C 0} C_DIS
LIN {X 47.61, Y 36.49, Z 12.0, A 0, B 90, C 0} C_DIS
LIN {X 45.69, Y 38.89, Z 12.0, A 0, B 90, C 0} C_DIS
LIN {X 45.17, Y 39.46, Z 12.0, A 0, B 90, C 0} C_DIS
LIN {X 43.1, Y 41.74, Z 12.0, A 0, B 90, C 0} C_DIS
LIN {X 42.55, Y 42.28, Z 12.0, A 0, B 90, C 0} C_DIS
LIN {X 40.34, Y 44.42, Z 12.0, A 0, B 90, C 0} C_DIS
LIN {X 39.75, Y 44.92, Z 12.0, A 0, B 90, C 0} C_DIS
LIN {X 37.41, Y 46.91, Z 12.0, A 0, B 90, C 0} C_DIS
LIN {X 36.79, Y 47.37, Z 12.0, A 0, B 90, C 0} C_DIS
LIN {X 34.33, Y 49.21, Z 12.0, A 0, B 90, C 0} C_DIS
LIN {X 33.68, Y 49.63, Z 12.0, A 0, B 90, C 0} C_DIS
LIN {X 31.1, Y 51.31, Z 12.0, A 0, B 90, C 0} C_DIS
LIN {X 30.43, Y 51.69, Z 12.0, A 0, B 90, C 0} C_DIS
LIN {X 27.75, Y 53.2, Z 12.0, A 0, B 90, C 0} C_DIS
LIN {X 27.06, Y 53.53, Z 12.0, A 0, B 90, C 0} C_DIS
LIN {X 24.29, Y 54.86, Z 12.0, A 0, B 90, C 0} C_DIS
LIN {X 23.57, Y 55.15, Z 12.0, A 0, B 90, C 0} C_DIS
LIN {X 20.72, Y 56.31, Z 12.0, A 0, B 90, C 0} C_DIS
LIN {X 19.99, Y 56.55, Z 12.0, A 0, B 90, C 0} C_DIS
LIN {X 17.07, Y 57.52, Z 12.0, A 0, B 90, C 0} C_DIS
LIN {X 16.33, Y 57.72, Z 12.0, A 0, B 90, C 0} C_DIS
LIN {X 13.35, Y 58.5, Z 12.0, A 0, B 90, C 0} C_DIS
LIN {X 12.6, Y 58.64, Z 12.0, A 0, B 90, C 0} C_DIS
LIN {X 9.58, Y 59.23, Z 12.0, A 0, B 90, C 0} C_DIS
LIN {X 8.81, Y 59.33, Z 12.0, A 0, B 90, C 0} C_DIS
LIN {X 5.76, Y 59.72, Z 12.0, A 0, B 90, C 0} C_DIS
LIN {X 4.99, Y 59.77, Z 12.0, A 0, B 90, C 0} C_DIS
LIN {X 1.92, Y 59.97, Z 12.0, A 0, B 90, C 0} C_DIS
LIN {X 1.15, Y 59.97, Z 12.0, A 0, B 90, C 0} C_DIS
LIN {X -1.92, Y 59.97, Z 12.0, A 0, B 90, C 0} C_DIS
LIN {X -2.69, Y 59.92, Z 12.0, A 0, B 90, C 0} C_DIS
LIN {X -5.76, Y 59.72, Z 12.0, A 0, B 90, C 0} C_DIS
LIN {X -6.52, Y 59.62, Z 12.0, A 0, B 90, C 0} C_DIS
LIN {X -9.58, Y 59.23, Z 12.0, A 0, B 90, C 0} C_DIS
LIN {X -10.33, Y 59.08, Z 12.0, A 0, B 90, C 0} C_DIS
LIN {X -13.35, Y 58.5, Z 12.0, A 0, B 90, C 0} C_DIS
LIN {X -14.1, Y 58.3, Z 12.0, A 0, B 90, C 0} C_DIS
LIN {X -17.07, Y 57.52, Z 12.0, A 0, B 90, C 0} C_DIS
LIN {X -17.8, Y 57.28, Z 12.0, A 0, B 90, C 0} C_DIS
LIN {X -20.72, Y 56.31, Z 12.0, A 0, B 90, C 0} C_DIS
LIN {X -21.43, Y 56.02, Z 12.0, A 0, B 90, C 0} C_DIS
LIN {X -24.29, Y 54.86, Z 12.0, A 0, B 90, C 0} C_DIS
LIN {X -24.98, Y 54.53, Z 12.0, A 0, B 90, C 0} C_DIS
LIN {X -27.75, Y 53.2, Z 12.0, A 0, B 90, C 0} C_DIS
LIN {X -28.42, Y 52.82, Z 12.0, A 0, B 90, C 0} C_DIS
LIN {X -31.1, Y 51.31, Z 12.0, A 0, B 90, C 0} C_DIS
LIN {X -31.75, Y 50.89, Z 12.0, A 0, B 90, C 0} C_DIS
LIN {X -34.33, Y 49.21, Z 12.0, A 0, B 90, C 0} C_DIS
LIN {X -34.94, Y 48.75, Z 12.0, A 0, B 90, C 0} C_DIS
LIN {X -37.41, Y 46.91, Z 12.0, A 0, B 90, C 0} C_DIS
LIN {X -38.0, Y 46.41, Z 12.0, A 0, B 90, C 0} C_DIS
LIN {X -40.34, Y 44.42, Z 12.0, A 0, B 90, C 0} C_DIS
LIN {X -40.89, Y 43.88, Z 12.0, A 0, B 90, C 0} C_DIS
LIN {X -43.1, Y 41.74, Z 12.0, A 0, B 90, C 0} C_DIS
LIN {X -43.62, Y 41.17, Z 12.0, A 0, B 90, C 0} C_DIS
LIN {X -45.69, Y 38.89, Z 12.0, A 0, B 90, C 0} C_DIS
LIN {X -46.17, Y 38.29, Z 12.0, A 0, B 90, C 0} C_DIS
LIN {X -48.08, Y 35.89, Z 12.0, A 0, B 90, C 0} C_DIS
LIN {X -48.52, Y 35.26, Z 12.0, A 0, B 90, C 0} C_DIS
LIN {X -50.29, Y 32.73, Z 12.0, A 0, B 90, C 0} C_DIS
LIN {X -50.68, Y 32.07, Z 12.0, A 0, B 90, C 0} C_DIS
LIN {X -52.28, Y 29.44, Z 12.0, A 0, B 90, C 0} C_DIS
LIN {X -52.63, Y 28.76, Z 12.0, A 0, B 90, C 0} C_DIS
LIN {X -54.06, Y 26.03, Z 12.0, A 0, B 90, C 0} C_DIS
LIN {X -54.37, Y 25.33, Z 12.0, A 0, B 90, C 0} C_DIS
LIN {X -55.62, Y 22.52, Z 12.0, A 0, B 90, C 0} C_DIS
LIN {X -55.88, Y 21.79, Z 12.0, A 0, B 90, C 0} C_DIS
LIN {X -56.94, Y 18.91, Z 12.0, A 0, B 90, C 0} C_DIS
LIN {X -57.16, Y 18.17, Z 12.0, A 0, B 90, C 0} C_DIS
LIN {X -58.04, Y 15.22, Z 12.0, A 0, B 90, C 0} C_DIS
LIN {X -58.21, Y 14.47, Z 12.0, A 0, B 90, C 0} C_DIS
LIN {X -58.89, Y 11.47, Z 12.0, A 0, B 90, C 0} C_DIS
LIN {X -59.02, Y 10.71, Z 12.0, A 0, B 90, C 0} C_DIS
LIN {X -59.51, Y 7.67, Z 12.0, A 0, B 90, C 0} C_DIS
LIN {X -59.58, Y 6.91, Z 12.0, A 0, B 90, C 0} C_DIS
LIN {X -59.88, Y 3.84, Z 12.0, A 0, B 90, C 0} C_DIS
LIN {X -59.9, Y 3.08, Z 12.0, A 0, B 90, C 0} C_DIS
LIN {X -60.0, Y -0.0, Z 12.0, A 0, B 90, C 0} C_DIS
LIN {X -59.98, Y -0.77, Z 12.0, A 0, B 90, C 0} C_DIS
LIN {X -59.88, Y -3.84, Z 12.0, A 0, B 90, C 0} C_DIS
LIN {X -59.8, Y -4.61, Z 12.0, A 0, B 90, C 0} C_DIS
LIN {X -59.51, Y -7.67, Z 12.0, A 0, B 90, C 0} C_DIS
LIN {X -59.38, Y -8.43, Z 12.0, A 0, B 90, C 0} C_DIS
LIN {X -58.89, Y -11.47, Z 12.0, A 0, B 90, C 0} C_DIS
LIN {X -58.72, Y -12.22, Z 12.0, A 0, B 90, C 0} C_DIS
LIN {X -58.04, Y -15.22, Z 12.0, A 0, B 90, C 0} C_DIS
LIN {X -57.82, Y -15.96, Z 12.0, A 0, B 90, C 0} C_DIS
LIN {X -56.94, Y -18.91, Z 12.0, A 0, B 90, C 0} C_DIS
LIN {X -56.68, Y -19.63, Z 12.0, A 0, B 90, C 0} C_DIS
LIN {X -55.62, Y -22.52, Z 12.0, A 0, B 90, C 0} C_DIS
LIN {X -55.3, Y -23.22, Z 12.0, A 0, B 90, C 0} C_DIS
LIN {X -54.06, Y -26.03, Z 12.0, A 0, B 90, C 0} C_DIS
LIN {X -53.7, Y -26.72, Z 12.0, A 0, B 90, C 0} C_DIS
LIN {X -52.28, Y -29.44, Z 12.0, A 0, B 90, C 0} C_DIS
LIN {X -51.88, Y -30.1, Z 12.0, A 0, B 90, C 0} C_DIS
LIN {X -50.29, Y -32.73, Z 12.0, A 0, B 90, C 0} C_DIS
LIN {X -49.85, Y -33.36, Z 12.0, A 0, B 90, C 0} C_DIS
LIN {X -48.08, Y -35.89, Z 12.0, A 0, B 90, C 0} C_DIS
LIN {X -47.61, Y -36.49, Z 12.0, A 0, B 90, C 0} C_DIS
LIN {X -45.69, Y -38.89, Z 12.0, A 0, B 90, C 0} C_DIS
LIN {X -45.17, Y -39.46, Z 12.0, A 0, B 90, C 0} C_DIS
LIN {X -43.1, Y -41.74, Z 12.0, A 0, B 90, C 0} C_DIS
LIN {X -42.55, Y -42.28, Z 12.0, A 0, B 90, C 0} C_DIS
LIN {X -40.34, Y -44.42, Z 12.0, A 0, B 90, C 0} C_DIS
LIN {X -39.75, Y -44.92, Z 12.0, A 0, B 90, C 0} C_DIS
LIN {X -37.41, Y -46.91, Z 12.0, A 0, B 90, C 0} C_DIS
LIN {X -36.79, Y -47.37, Z 12.0, A 0, B 90, C 0} C_DIS
$OUT[1] = FALSE

; END LAYER 5
LIN {X -34.33, Y -49.21, Z 12.0, A 0, B 90, C 0} C_DIS
WAIT SEC 3
LIN {X -34.33, Y -49.21, Z 14.0, A 0, B 90, C 0} C_DIS
$OUT[1] = TRUE
WAIT SEC 0.8
LIN {X -34.33, Y -49.21, Z 14.0, A 0, B 90, C 0} C_DIS
LIN {X -34.33, Y -49.21, Z 14.0, A 0, B 90, C 0} C_DIS
LIN {X -33.55, Y -49.71, Z 14.0, A 0, B 90, C 0} C_DIS
LIN {X -31.1, Y -51.31, Z 14.0, A 0, B 90, C 0} C_DIS
LIN {X -30.3, Y -51.76, Z 14.0, A 0, B 90, C 0} C_DIS
LIN {X -27.75, Y -53.2, Z 14.0, A 0, B 90, C 0} C_DIS
LIN {X -26.92, Y -53.6, Z 14.0, A 0, B 90, C 0} C_DIS
LIN {X -24.29, Y -54.86, Z 14.0, A 0, B 90, C 0} C_DIS
LIN {X -23.43, Y -55.21, Z 14.0, A 0, B 90, C 0} C_DIS
LIN {X -20.72, Y -56.31, Z 14.0, A 0, B 90, C 0} C_DIS
LIN {X -19.85, Y -56.6, Z 14.0, A 0, B 90, C 0} C_DIS
LIN {X -17.07, Y -57.52, Z 14.0, A 0, B 90, C 0} C_DIS
LIN {X -16.18, Y -57.75, Z 14.0, A 0, B 90, C 0} C_DIS
LIN {X -13.35, Y -58.5, Z 14.0, A 0, B 90, C 0} C_DIS
LIN {X -12.45, Y -58.67, Z 14.0, A 0, B 90, C 0} C_DIS
LIN {X -9.58, Y -59.23, Z 14.0, A 0, B 90, C 0} C_DIS
LIN {X -8.66, Y -59.35, Z 14.0, A 0, B 90, C 0} C_DIS
LIN {X -5.76, Y -59.72, Z 14.0, A 0, B 90, C 0} C_DIS
LIN {X -4.84, Y -59.78, Z 14.0, A 0, B 90, C 0} C_DIS
LIN {X -1.92, Y -59.97, Z 14.0, A 0, B 90, C 0} C_DIS
LIN {X -1.0, Y -59.97, Z 14.0, A 0, B 90, C 0} C_DIS
LIN {X 1.92, Y -59.97, Z 14.0, A 0, B 90, C 0} C_DIS
LIN {X 2.84, Y -59.91, Z 14.0, A 0, B 90, C 0} C_DIS
LIN {X 5.76, Y -59.72, Z 14.0, A 0, B 90, C 0} C_DIS
LIN {X 6.68, Y -59.6, Z 14.0, A 0, B 90, C 0} C_DIS
LIN {X 9.58, Y -59.23, Z 14.0, A 0, B 90, C 0} C_DIS
LIN {X 10.48, Y -59.05, Z 14.0, A 0, B 90, C 0} C_DIS
LIN {X 13.35, Y -58.5, Z 14.0, A 0, B 90, C 0} C_DIS
LIN {X 14.24, Y -58.26, Z 14.0, A 0, B 90, C 0} C_DIS
LIN {X 17.07, Y -57.52, Z 14.0, A 0, B 90, C 0} C_DIS
LIN {X 17.95, Y -57.23, Z 14.0, A 0, B 90, C 0} C_DIS
LIN {X 20.72, Y -56.31, Z 14.0, A 0, B 90, C 0} C_DIS
LIN {X 21.58, Y -55.96, Z 14.0, A 0, B 90, C 0} C_DIS
LIN {X 24.29, Y -54.86, Z 14.0, A 0, B 90, C 0} C_DIS
LIN {X 25.12, Y -54.46, Z 14.0, A 0, B 90, C 0} C_DIS
LIN {X 27.75, Y -53.2, Z 14.0, A 0, B 90, C 0} C_DIS
LIN {X 28.56, Y -52.74, Z 14.0, A 0, B 90, C 0} C_DIS
LIN {X 31.1, Y -51.31, Z 14.0, A 0, B 90, C 0} C_DIS
LIN {X 31.88, Y -50.8, Z 14.0, A 0, B 90, C 0} C_DIS
LIN {X 34.33, Y -49.21, Z 14.0, A 0, B 90, C 0} C_DIS
LIN {X 35.07, Y -48.66, Z 14.0, A 0, B 90, C 0} C_DIS
LIN {X 37.41, Y -46.91, Z 14.0, A 0, B 90, C 0} C_DIS
LIN {X 38.11, Y -46.31, Z 14.0, A 0, B 90, C 0} C_DIS
LIN {X 40.34, Y -44.42, Z 14.0, A 0, B 90, C 0} C_DIS
LIN {X 41.0, Y -43.77, Z 14.0, A 0, B 90, C 0} C_DIS
LIN {X 43.1, Y -41.74, Z 14.0, A 0, B 90, C 0} C_DIS
LIN {X 43.72, Y -41.06, Z 14.0, A 0, B 90, C 0} C_DIS
LIN {X 45.69, Y -38.89, Z 14.0, A 0, B 90, C 0} C_DIS
LIN {X 46.26, Y -38.17, Z 14.0, A 0, B 90, C 0} C_DIS
LIN {X 48.08, Y -35.89, Z 14.0, A 0, B 90, C 0} C_DIS
LIN {X 48.61, Y -35.13, Z 14.0, A 0, B 90, C 0} C_DIS
LIN {X 50.29, Y -32.73, Z 14.0, A 0, B 90, C 0} C_DIS
LIN {X 50.76, Y -31.94, Z 14.0, A 0, B 90, C 0} C_DIS
LIN {X 52.28, Y -29.44, Z 14.0, A 0, B 90, C 0} C_DIS
LIN {X 52.71, Y -28.62, Z 14.0, A 0, B 90, C 0} C_DIS
LIN {X 54.06, Y -26.03, Z 14.0, A 0, B 90, C 0} C_DIS
LIN {X 54.43, Y -25.19, Z 14.0, A 0, B 90, C 0} C_DIS
LIN {X 55.62, Y -22.52, Z 14.0, A 0, B 90, C 0} C_DIS
LIN {X 55.93, Y -21.65, Z 14.0, A 0, B 90, C 0} C_DIS
LIN {X 56.94, Y -18.91, Z 14.0, A 0, B 90, C 0} C_DIS
LIN {X 57.21, Y -18.02, Z 14.0, A 0, B 90, C 0} C_DIS
LIN {X 58.04, Y -15.22, Z 14.0, A 0, B 90, C 0} C_DIS
LIN {X 58.24, Y -14.32, Z 14.0, A 0, B 90, C 0} C_DIS
LIN {X 58.89, Y -11.47, Z 14.0, A 0, B 90, C 0} C_DIS
LIN {X 59.04, Y -10.56, Z 14.0, A 0, B 90, C 0} C_DIS
LIN {X 59.51, Y -7.67, Z 14.0, A 0, B 90, C 0} C_DIS
LIN {X 59.6, Y -6.75, Z 14.0, A 0, B 90, C 0} C_DIS
LIN {X 59.88, Y -3.84, Z 14.0, A 0, B 90, C 0} C_DIS
LIN {X 59.91, Y -2.92, Z 14.0, A 0, B 90, C 0} C_DIS
LIN {X 60.0, Y 0.0, Z 14.0, A 0, B 90, C 0} C_DIS
LIN {X 59.97, Y 0.92, Z 14.0, A 0, B 90, C 0} C_DIS
LIN {X 59.88, Y 3.84, Z 14.0, A 0, B 90, C 0} C_DIS
LIN {X 59.79, Y 4.76, Z 14.0, A 0, B 90, C 0} C_DIS
LIN {X 59.51, Y 7.67, Z 14.0, A 0, B 90, C 0} C_DIS
LIN {X 59.36, Y 8.58, Z 14.0, A 0, B 90, C 0} C_DIS
LIN {X 58.89, Y 11.47, Z 14.0, A 0, B 90, C 0} C_DIS
LIN {X 58.69, Y 12.37, Z 14.0, A 0, B 90, C 0} C_DIS
LIN {X 58.04, Y 15.22, Z 14.0, A 0, B 90, C 0} C_DIS
LIN {X 57.78, Y 16.1, Z 14.0, A 0, B 90, C 0} C_DIS
LIN {X 56.94, Y 18.91, Z 14.0, A 0, B 90, C 0} C_DIS
LIN {X 56.62, Y 19.77, Z 14.0, A 0, B 90, C 0} C_DIS
LIN {X 55.62, Y 22.52, Z 14.0, A 0, B 90, C 0} C_DIS
LIN {X 55.24, Y 23.36, Z 14.0, A 0, B 90, C 0} C_DIS
LIN {X 54.06, Y 26.03, Z 14.0, A 0, B 90, C 0} C_DIS
LIN {X 53.63, Y 26.85, Z 14.0, A 0, B 90, C 0} C_DIS
LIN {X 52.28, Y 29.44, Z 14.0, A 0, B 90, C 0} C_DIS
LIN {X 51.8, Y 30.23, Z 14.0, A 0, B 90, C 0} C_DIS
LIN {X 50.29, Y 32.73, Z 14.0, A 0, B 90, C 0} C_DIS
LIN {X 49.76, Y 33.49, Z 14.0, A 0, B 90, C 0} C_DIS
LIN {X 48.08, Y 35.89, Z 14.0, A 0, B 90, C 0} C_DIS
LIN {X 47.51, Y 36.61, Z 14.0, A 0, B 90, C 0} C_DIS
LIN {X 45.69, Y 38.89, Z 14.0, A 0, B 90, C 0} C_DIS
LIN {X 45.07, Y 39.58, Z 14.0, A 0, B 90, C 0} C_DIS
LIN {X 43.1, Y 41.74, Z 14.0, A 0, B 90, C 0} C_DIS
LIN {X 42.44, Y 42.38, Z 14.0, A 0, B 90, C 0} C_DIS
LIN {X 40.34, Y 44.42, Z 14.0, A 0, B 90, C 0} C_DIS
LIN {X 39.64, Y 45.02, Z 14.0, A 0, B 90, C 0} C_DIS
LIN {X 37.41, Y 46.91, Z 14.0, A 0, B 90, C 0} C_DIS
LIN {X 36.67, Y 47.46, Z 14.0, A 0, B 90, C 0} C_DIS
LIN {X 34.33, Y 49.21, Z 14.0, A 0, B 90, C 0} C_DIS
LIN {X 33.55, Y 49.71, Z 14.0, A 0, B 90, C 0} C_DIS
LIN {X 31.1, Y 51.31, Z 14.0, A 0, B 90, C 0} C_DIS
LIN {X 30.3, Y 51.76, Z 14.0, A 0, B 90, C 0} C_DIS
LIN {X 27.75, Y 53.2, Z 14.0, A 0, B 90, C 0} C_DIS
LIN {X 26.92, Y 53.6, Z 14.0, A 0, B 90, C 0} C_DIS
LIN {X 24.29, Y 54.86, Z 14.0, A 0, B 90, C 0} C_DIS
LIN {X 23.43, Y 55.21, Z 14.0, A 0, B 90, C 0} C_DIS
LIN {X 20.72, Y 56.31, Z 14.0, A 0, B 90, C 0} C_DIS
LIN {X 19.85, Y 56.6, Z 14.0, A 0, B 90, C 0} C_DIS
LIN {X 17.07, Y 57.52, Z 14.0, A 0, B 90, C 0} C_DIS
LIN {X 16.18, Y 57.75, Z 14.0, A 0, B 90, C 0} C_DIS
LIN {X 13.35, Y 58.5, Z 14.0, A 0, B 90, C 0} C_DIS
LIN {X 12.45, Y 58.67, Z 14.0, A 0, B 90, C 0} C_DIS
LIN {X 9.58, Y 59.23, Z 14.0, A 0, B 90, C 0} C_DIS
LIN {X 8.66, Y 59.35, Z 14.0, A 0, B 90, C 0} C_DIS
LIN {X 5.76, Y 59.72, Z 14.0, A 0, B 90, C 0} C_DIS
LIN {X 4.84, Y 59.78, Z 14.0, A 0, B 90, C 0} C_DIS
LIN {X 1.92, Y 59.97, Z 14.0, A 0, B 90, C 0} C_DIS
LIN {X 1.0, Y 59.97, Z 14.0, A 0, B 90, C 0} C_DIS
LIN {X -1.92, Y 59.97, Z 14.0, A 0, B 90, C 0} C_DIS
LIN {X -2.84, Y 59.91, Z 14.0, A 0, B 90, C 0} C_DIS
LIN {X -5.76, Y 59.72, Z 14.0, A 0, B 90, C 0} C_DIS
LIN {X -6.68, Y 59.6, Z 14.0, A 0, B 90, C 0} C_DIS
LIN {X -9.58, Y 59.23, Z 14.0, A 0, B 90, C 0} C_DIS
LIN {X -10.48, Y 59.05, Z 14.0, A 0, B 90, C 0} C_DIS
LIN {X -13.35, Y 58.5, Z 14.0, A 0, B 90, C 0} C_DIS
LIN {X -14.24, Y 58.26, Z 14.0, A 0, B 90, C 0} C_DIS
LIN {X -17.07, Y 57.52, Z 14.0, A 0, B 90, C 0} C_DIS
LIN {X -17.95, Y 57.23, Z 14.0, A 0, B 90, C 0} C_DIS
LIN {X -20.72, Y 56.31, Z 14.0, A 0, B 90, C 0} C_DIS
LIN {X -21.58, Y 55.96, Z 14.0, A 0, B 90, C 0} C_DIS
LIN {X -24.29, Y 54.86, Z 14.0, A 0, B 90, C 0} C_DIS
LIN {X -25.12, Y 54.46, Z 14.0, A 0, B 90, C 0} C_DIS
LIN {X -27.75, Y 53.2, Z 14.0, A 0, B 90, C 0} C_DIS
LIN {X -28.56, Y 52.74, Z 14.0, A 0, B 90, C 0} C_DIS
LIN {X -31.1, Y 51.31, Z 14.0, A 0, B 90, C 0} C_DIS
LIN {X -31.88, Y 50.8, Z 14.0, A 0, B 90, C 0} C_DIS
LIN {X -34.33, Y 49.21, Z 14.0, A 0, B 90, C 0} C_DIS
LIN {X -35.07, Y 48.66, Z 14.0, A 0, B 90, C 0} C_DIS
LIN {X -37.41, Y 46.91, Z 14.0, A 0, B 90, C 0} C_DIS
LIN {X -38.11, Y 46.31, Z 14.0, A 0, B 90, C 0} C_DIS
LIN {X -40.34, Y 44.42, Z 14.0, A 0, B 90, C 0} C_DIS
LIN {X -41.0, Y 43.77, Z 14.0, A 0, B 90, C 0} C_DIS
LIN {X -43.1, Y 41.74, Z 14.0, A 0, B 90, C 0} C_DIS
LIN {X -43.72, Y 41.06, Z 14.0, A 0, B 90, C 0} C_DIS
LIN {X -45.69, Y 38.89, Z 14.0, A 0, B 90, C 0} C_DIS
LIN {X -46.26, Y 38.17, Z 14.0, A 0, B 90, C 0} C_DIS
LIN {X -48.08, Y 35.89, Z 14.0, A 0, B 90, C 0} C_DIS
LIN {X -48.61, Y 35.13, Z 14.0, A 0, B 90, C 0} C_DIS
LIN {X -50.29, Y 32.73, Z 14.0, A 0, B 90, C 0} C_DIS
LIN {X -50.76, Y 31.94, Z 14.0, A 0, B 90, C 0} C_DIS
LIN {X -52.28, Y 29.44, Z 14.0, A 0, B 90, C 0} C_DIS
LIN {X -52.71, Y 28.62, Z 14.0, A 0, B 90, C 0} C_DIS
LIN {X -54.06, Y 26.03, Z 14.0, A 0, B 90, C 0} C_DIS
LIN {X -54.43, Y 25.19, Z 14.0, A 0, B 90, C 0} C_DIS
LIN {X -55.62, Y 22.52, Z 14.0, A 0, B 90, C 0} C_DIS
LIN {X -55.93, Y 21.65, Z 14.0, A 0, B 90, C 0} C_DIS
LIN {X -56.94, Y 18.91, Z 14.0, A 0, B 90, C 0} C_DIS
LIN {X -57.21, Y 18.02, Z 14.0, A 0, B 90, C 0} C_DIS
LIN {X -58.04, Y 15.22, Z 14.0, A 0, B 90, C 0} C_DIS
LIN {X -58.24, Y 14.32, Z 14.0, A 0, B 90, C 0} C_DIS
LIN {X -58.89, Y 11.47, Z 14.0, A 0, B 90, C 0} C_DIS
LIN {X -59.04, Y 10.56, Z 14.0, A 0, B 90, C 0} C_DIS
LIN {X -59.51, Y 7.67, Z 14.0, A 0, B 90, C 0} C_DIS
LIN {X -59.6, Y 6.75, Z 14.0, A 0, B 90, C 0} C_DIS
LIN {X -59.88, Y 3.84, Z 14.0, A 0, B 90, C 0} C_DIS
LIN {X -59.91, Y 2.92, Z 14.0, A 0, B 90, C 0} C_DIS
LIN {X -60.0, Y -0.0, Z 14.0, A 0, B 90, C 0} C_DIS
LIN {X -59.97, Y -0.92, Z 14.0, A 0, B 90, C 0} C_DIS
LIN {X -59.88, Y -3.84, Z 14.0, A 0, B 90, C 0} C_DIS
LIN {X -59.79, Y -4.76, Z 14.0, A 0, B 90, C 0} C_DIS
LIN {X -59.51, Y -7.67, Z 14.0, A 0, B 90, C 0} C_DIS
LIN {X -59.36, Y -8.58, Z 14.0, A 0, B 90, C 0} C_DIS
LIN {X -58.89, Y -11.47, Z 14.0, A 0, B 90, C 0} C_DIS
LIN {X -58.69, Y -12.37, Z 14.0, A 0, B 90, C 0} C_DIS
LIN {X -58.04, Y -15.22, Z 14.0, A 0, B 90, C 0} C_DIS
LIN {X -57.78, Y -16.1, Z 14.0, A 0, B 90, C 0} C_DIS
LIN {X -56.94, Y -18.91, Z 14.0, A 0, B 90, C 0} C_DIS
LIN {X -56.62, Y -19.77, Z 14.0, A 0, B 90, C 0} C_DIS
LIN {X -55.62, Y -22.52, Z 14.0, A 0, B 90, C 0} C_DIS
LIN {X -55.24, Y -23.36, Z 14.0, A 0, B 90, C 0} C_DIS
LIN {X -54.06, Y -26.03, Z 14.0, A 0, B 90, C 0} C_DIS
LIN {X -53.63, Y -26.85, Z 14.0, A 0, B 90, C 0} C_DIS
LIN {X -52.28, Y -29.44, Z 14.0, A 0, B 90, C 0} C_DIS
LIN {X -51.8, Y -30.23, Z 14.0, A 0, B 90, C 0} C_DIS
LIN {X -50.29, Y -32.73, Z 14.0, A 0, B 90, C 0} C_DIS
LIN {X -49.76, Y -33.49, Z 14.0, A 0, B 90, C 0} C_DIS
LIN {X -48.08, Y -35.89, Z 14.0, A 0, B 90, C 0} C_DIS
LIN {X -47.51, Y -36.61, Z 14.0, A 0, B 90, C 0} C_DIS
LIN {X -45.69, Y -38.89, Z 14.0, A 0, B 90, C 0} C_DIS
LIN {X -45.07, Y -39.58, Z 14.0, A 0, B 90, C 0} C_DIS
LIN {X -43.1, Y -41.74, Z 14.0, A 0, B 90, C 0} C_DIS
LIN {X -42.44, Y -42.38, Z 14.0, A 0, B 90, C 0} C_DIS
LIN {X -40.34, Y -44.42, Z 14.0, A 0, B 90, C 0} C_DIS
LIN {X -39.64, Y -45.02, Z 14.0, A 0, B 90, C 0} C_DIS
LIN {X -37.41, Y -46.91, Z 14.0, A 0, B 90, C 0} C_DIS
LIN {X -36.67, Y -47.46, Z 14.0, A 0, B 90, C 0} C_DIS
$OUT[1] = FALSE

; END LAYER 6
LIN {X -34.33, Y -49.21, Z 14.0, A 0, B 90, C 0} C_DIS
WAIT SEC 3
LIN {X -34.33, Y -49.21, Z 16.0, A 0, B 90, C 0} C_DIS
$OUT[1] = TRUE
WAIT SEC 0.8
LIN {X -34.33, Y -49.21, Z 16.0, A 0, B 90, C 0} C_DIS
LIN {X -34.33, Y -49.21, Z 16.0, A 0, B 90, C 0} C_DIS
LIN {X -33.42, Y -49.8, Z 16.0, A 0, B 90, C 0} C_DIS
LIN {X -31.1, Y -51.31, Z 16.0, A 0, B 90, C 0} C_DIS
LIN {X -30.17, Y -51.84, Z 16.0, A 0, B 90, C 0} C_DIS
LIN {X -27.75, Y -53.2, Z 16.0, A 0, B 90, C 0} C_DIS
LIN {X -26.78, Y -53.66, Z 16.0, A 0, B 90, C 0} C_DIS
LIN {X -24.29, Y -54.86, Z 16.0, A 0, B 90, C 0} C_DIS
LIN {X -23.29, Y -55.27, Z 16.0, A 0, B 90, C 0} C_DIS
LIN {X -20.72, Y -56.31, Z 16.0, A 0, B 90, C 0} C_DIS
LIN {X -19.7, Y -56.65, Z 16.0, A 0, B 90, C 0} C_DIS
LIN {X -17.07, Y -57.52, Z 16.0, A 0, B 90, C 0} C_DIS
LIN {X -16.03, Y -57.79, Z 16.0, A 0, B 90, C 0} C_DIS
LIN {X -13.35, Y -58.5, Z 16.0, A 0, B 90, C 0} C_DIS
LIN {X -12.29, Y -58.7, Z 16.0, A 0, B 90, C 0} C_DIS
LIN {X -9.58, Y -59.23, Z 16.0, A 0, B 90, C 0} C_DIS
LIN {X -8.51, Y -59.37, Z 16.0, A 0, B 90, C 0} C_DIS
LIN {X -5.76, Y -59.72, Z 16.0, A 0, B 90, C 0} C_DIS
LIN {X -4.69, Y -59.79, Z 16.0, A 0, B 90, C 0} C_DIS
LIN {X -1.92, Y -59.97, Z 16.0, A 0, B 90, C 0} C_DIS
LIN {X -0.85, Y -59.97, Z 16.0, A 0, B 90, C 0} C_DIS
LIN {X 1.92, Y -59.97, Z 16.0, A 0, B 90, C 0} C_DIS
LIN {X 3.0, Y -59.9, Z 16.0, A 0, B 90, C 0} C_DIS
LIN {X 5.76, Y -59.72, Z 16.0, A 0, B 90, C 0} C_DIS
LIN {X 6.83, Y -59.59, Z 16.0, A 0, B 90, C 0} C_DIS
LIN {X 9.58, Y -59.23, Z 16.0, A 0, B 90, C 0} C_DIS
LIN {X 10.63, Y -59.03, Z 16.0, A 0, B 90, C 0} C_DIS
LIN {X 13.35, Y -58.5, Z 16.0, A 0, B 90, C 0} C_DIS
LIN {X 14.39, Y -58.22, Z 16.0, A 0, B 90, C 0} C_DIS
LIN {X 17.07, Y -57.52, Z 16.0, A 0, B 90, C 0} C_DIS
LIN {X 18.09, Y -57.18, Z 16.0, A 0, B 90, C 0} C_DIS
LIN {X 20.72, Y -56.31, Z 16.0, A 0, B 90, C 0} C_DIS
LIN {X 21.72, Y -55.9, Z 16.0, A 0, B 90, C 0} C_DIS
LIN {X 24.29, Y -54.86, Z 16.0, A 0, B 90, C 0} C_DIS
LIN {X 25.26, Y -54.4, Z 16.0, A 0, B 90, C 0} C_DIS
LIN {X 27.75, Y -53.2, Z 16.0, A 0, B 90, C 0} C_DIS
LIN {X 28.69, Y -52.67, Z 16.0, A 0, B 90, C 0} C_DIS
LIN {X 31.1, Y -51.31, Z 16.0, A 0, B 90, C 0} C_DIS
LIN {X 32.01, Y -50.72, Z 16.0, A 0, B 90, C 0} C_DIS
LIN {X 34.33, Y -49.21, Z 16.0, A 0, B 90, C 0} C_DIS
LIN {X 35.19, Y -48.57, Z 16.0, A 0, B 90, C 0} C_DIS
LIN {X 37.41, Y -46.91, Z 16.0, A 0, B 90, C 0} C_DIS
LIN {X 38.23, Y -46.21, Z 16.0, A 0, B 90, C 0} C_DIS
LIN {X 40.34, Y -44.42, Z 16.0, A 0, B 90, C 0} C_DIS
LIN {X 41.11, Y -43.67, Z 16.0, A 0, B 90, C 0} C_DIS
LIN {X 43.1, Y -41.74, Z 16.0, A 0, B 90, C 0} C_DIS
LIN {X 43.82, Y -40.94, Z 16.0, A 0, B 90, C 0} C_DIS
LIN {X 45.69, Y -38.89, Z 16.0, A 0, B 90, C 0} C_DIS
LIN {X 46.36, Y -38.05, Z 16.0, A 0, B 90, C 0} C_DIS
LIN {X 48.08, Y -35.89, Z 16.0, A 0, B 90, C 0} C_DIS
LIN {X 48.7, Y -35.0, Z 16.0, A 0, B 90, C 0} C_DIS
LIN {X 50.29, Y -32.73, Z 16.0, A 0, B 90, C 0} C_DIS
LIN {X 50.84, Y -31.81, Z 16.0, A 0, B 90, C 0} C_DIS
LIN {X 52.28, Y -29.44, Z 16.0, A 0, B 90, C 0} C_DIS
LIN {X 52.78, Y -28.49, Z 16.0, A 0, B 90, C 0} C_DIS
LIN {X 54.06, Y -26.03, Z 16.0, A 0, B 90, C 0} C_DIS
LIN {X 54.49, Y -25.05, Z 16.0, A 0, B 90, C 0} C_DIS
LIN {X 55.62, Y -22.52, Z 16.0, A 0, B 90, C 0} C_DIS
LIN {X 55.99, Y -21.51, Z 16.0, A 0, B 90, C 0} C_DIS
LIN {X 56.94, Y -18.91, Z 16.0, A 0, B 90, C 0} C_DIS
LIN {X 57.25, Y -17.87, Z 16.0, A 0, B 90, C 0} C_DIS
LIN {X 58.04, Y -15.22, Z 16.0, A 0, B 90, C 0} C_DIS
LIN {X 58.28, Y -14.17, Z 16.0, A 0, B 90, C 0} C_DIS
LIN {X 58.89, Y -11.47, Z 16.0, A 0, B 90, C 0} C_DIS
LIN {X 59.07, Y -10.41, Z 16.0, A 0, B 90, C 0} C_DIS
LIN {X 59.51, Y -7.67, Z 16.0, A 0, B 90, C 0} C_DIS
LIN {X 59.61, Y -6.6, Z 16.0, A 0, B 90, C 0} C_DIS
LIN {X 59.88, Y -3.84, Z 16.0, A 0, B 90, C 0} C_DIS
LIN {X 59.91, Y -2.77, Z 16.0, A 0, B 90, C 0} C_DIS
LIN {X 60.0, Y -0.0, Z 16.0, A 0, B 90, C 0} C_DIS
LIN {X 59.97, Y 1.08, Z 16.0, A 0, B 90, C 0} C_DIS
LIN {X 59.88, Y 3.84, Z 16.0, A 0, B 90, C 0} C_DIS
LIN {X 59.77, Y 4.92, Z 16.0, A 0, B 90, C 0} C_DIS
LIN {X 59.51, Y 7.67, Z 16.0, A 0, B 90, C 0} C_DIS
LIN {X 59.34, Y 8.74, Z 16.0, A 0, B 90, C 0} C_DIS
LIN {X 58.89, Y 11.47, Z 16.0, A 0, B 90, C 0} C_DIS
LIN {X 58.65, Y 12.52, Z 16.0, A 0, B 90, C 0} C_DIS
LIN {X 58.04, Y 15.22, Z 16.0, A 0, B 90, C 0} C_DIS
LIN {X 57.73, Y 16.25, Z 16.0, A 0, B 90, C 0} C_DIS
LIN {X 56.94, Y 18.91, Z 16.0, A 0, B 90, C 0} C_DIS
LIN {X 56.57, Y 19.92, Z 16.0, A 0, B 90, C 0} C_DIS
LIN {X 55.62, Y 22.52, Z 16.0, A 0, B 90, C 0} C_DIS
LIN {X 55.18, Y 23.5, Z 16.0, A 0, B 90, C 0} C_DIS
LIN {X 54.06, Y 26.03, Z 16.0, A 0, B 90, C 0} C_DIS
LIN {X 53.56, Y 26.99, Z 16.0, A 0, B 90, C 0} C_DIS
LIN {X 52.28, Y 29.44, Z 16.0, A 0, B 90, C 0} C_DIS
LIN {X 51.72, Y 30.36, Z 16.0, A 0, B 90, C 0} C_DIS
LIN {X 50.29, Y 32.73, Z 16.0, A 0, B 90, C 0} C_DIS
LIN {X 49.67, Y 33.62, Z 16.0, A 0, B 90, C 0} C_DIS
LIN {X 48.08, Y 35.89, Z 16.0, A 0, B 90, C 0} C_DIS
LIN {X 47.41, Y 36.73, Z 16.0, A 0, B 90, C 0} C_DIS
LIN {X 45.69, Y 38.89, Z 16.0, A 0, B 90, C 0} C_DIS
LIN {X 44.96, Y 39.69, Z 16.0, A 0, B 90, C 0} C_DIS
LIN {X 43.1, Y 41.74, Z 16.0, A 0, B 90, C 0} C_DIS
LIN {X 42.33, Y 42.49, Z 16.0, A 0, B 90, C 0} C_DIS
LIN {X 40.34, Y 44.42, Z 16.0, A 0, B 90, C 0} C_DIS
LIN {X 39.52, Y 45.11, Z 16.0, A 0, B 90, C 0} C_DIS
LIN {X 37.41, Y 46.91, Z 16.0, A 0, B 90, C 0} C_DIS
LIN {X 36.55, Y 47.55, Z 16.0, A 0, B 90, C 0} C_DIS
LIN {X 34.33, Y 49.21, Z 16.0, A 0, B 90, C 0} C_DIS
LIN {X 33.42, Y 49.8, Z 16.0, A 0, B 90, C 0} C_DIS
LIN {X 31.1, Y 51.31, Z 16.0, A 0, B 90, C 0} C_DIS
LIN {X 30.17, Y 51.84, Z 16.0, A 0, B 90, C 0} C_DIS
LIN {X 27.75, Y 53.2, Z 16.0, A 0, B 90, C 0} C_DIS
LIN {X 26.78, Y 53.66, Z 16.0, A 0, B 90, C 0} C_DIS
LIN {X 24.29, Y 54.86, Z 16.0, A 0, B 90, C 0} C_DIS
LIN {X 23.29, Y 55.27, Z 16.0, A 0, B 90, C 0} C_DIS
LIN {X 20.72, Y 56.31, Z 16.0, A 0, B 90, C 0} C_DIS
LIN {X 19.7, Y 56.65, Z 16.0, A 0, B 90, C 0} C_DIS
LIN {X 17.07, Y 57.52, Z 16.0, A 0, B 90, C 0} C_DIS
LIN {X 16.03, Y 57.79, Z 16.0, A 0, B 90, C 0} C_DIS
LIN {X 13.35, Y 58.5, Z 16.0, A 0, B 90, C 0} C_DIS
LIN {X 12.29, Y 58.7, Z 16.0, A 0, B 90, C 0} C_DIS
LIN {X 9.58, Y 59.23, Z 16.0, A 0, B 90, C 0} C_DIS
LIN {X 8.51, Y 59.37, Z 16.0, A 0, B 90, C 0} C_DIS
LIN {X 5.76, Y 59.72, Z 16.0, A 0, B 90, C 0} C_DIS
LIN {X 4.69, Y 59.79, Z 16.0, A 0, B 90, C 0} C_DIS
LIN {X 1.92, Y 59.97, Z 16.0, A 0, B 90, C 0} C_DIS
LIN {X 0.85, Y 59.97, Z 16.0, A 0, B 90, C 0} C_DIS
LIN {X -1.92, Y 59.97, Z 16.0, A 0, B 90, C 0} C_DIS
LIN {X -3.0, Y 59.9, Z 16.0, A 0, B 90, C 0} C_DIS
LIN {X -5.76, Y 59.72, Z 16.0, A 0, B 90, C 0} C_DIS
LIN {X -6.83, Y 59.59, Z 16.0, A 0, B 90, C 0} C_DIS
LIN {X -9.58, Y 59.23, Z 16.0, A 0, B 90, C 0} C_DIS
LIN {X -10.63, Y 59.03, Z 16.0, A 0, B 90, C 0} C_DIS
LIN {X -13.35, Y 58.5, Z 16.0, A 0, B 90, C 0} C_DIS
LIN {X -14.39, Y 58.22, Z 16.0, A 0, B 90, C 0} C_DIS
LIN {X -17.07, Y 57.52, Z 16.0, A 0, B 90, C 0} C_DIS
LIN {X -18.09, Y 57.18, Z 16.0, A 0, B 90, C 0} C_DIS
LIN {X -20.72, Y 56.31, Z 16.0, A 0, B 90, C 0} C_DIS
LIN {X -21.72, Y 55.9, Z 16.0, A 0, B 90, C 0} C_DIS
LIN {X -24.29, Y 54.86, Z 16.0, A 0, B 90, C 0} C_DIS
LIN {X -25.26, Y 54.4, Z 16.0, A 0, B 90, C 0} C_DIS
LIN {X -27.75, Y 53.2, Z 16.0, A 0, B 90, C 0} C_DIS
LIN {X -28.69, Y 52.67, Z 16.0, A 0, B 90, C 0} C_DIS
LIN {X -31.1, Y 51.31, Z 16.0, A 0, B 90, C 0} C_DIS
LIN {X -32.01, Y 50.72, Z 16.0, A 0, B 90, C 0} C_DIS
LIN {X -34.33, Y 49.21, Z 16.0, A 0, B 90, C 0} C_DIS
LIN {X -35.19, Y 48.57, Z 16.0, A 0, B 90, C 0} C_DIS
LIN {X -37.41, Y 46.91, Z 16.0, A 0, B 90, C 0} C_DIS
LIN {X -38.23, Y 46.21, Z 16.0, A 0, B 90, C 0} C_DIS
LIN {X -40.34, Y 44.42, Z 16.0, A 0, B 90, C 0} C_DIS
LIN {X -41.11, Y 43.67, Z 16.0, A 0, B 90, C 0} C_DIS
LIN {X -43.1, Y 41.74, Z 16.0, A 0, B 90, C 0} C_DIS
LIN {X -43.82, Y 40.94, Z 16.0, A 0, B 90, C 0} C_DIS
LIN {X -45.69, Y 38.89, Z 16.0, A 0, B 90, C 0} C_DIS
LIN {X -46.36, Y 38.05, Z 16.0, A 0, B 90, C 0} C_DIS
LIN {X -48.08, Y 35.89, Z 16.0, A 0, B 90, C 0} C_DIS
LIN {X -48.7, Y 35.0, Z 16.0, A 0, B 90, C 0} C_DIS
LIN {X -50.29, Y 32.73, Z 16.0, A 0, B 90, C 0} C_DIS
LIN {X -50.84, Y 31.81, Z 16.0, A 0, B 90, C 0} C_DIS
LIN {X -52.28, Y 29.44, Z 16.0, A 0, B 90, C 0} C_DIS
LIN {X -52.78, Y 28.49, Z 16.0, A 0, B 90, C 0} C_DIS
LIN {X -54.06, Y 26.03, Z 16.0, A 0, B 90, C 0} C_DIS
LIN {X -54.49, Y 25.05, Z 16.0, A 0, B 90, C 0} C_DIS
LIN {X -55.62, Y 22.52, Z 16.0, A 0, B 90, C 0} C_DIS
LIN {X -55.99, Y 21.51, Z 16.0, A 0, B 90, C 0} C_DIS
LIN {X -56.94, Y 18.91, Z 16.0, A 0, B 90, C 0} C_DIS
LIN {X -57.25, Y 17.87, Z 16.0, A 0, B 90, C 0} C_DIS
LIN {X -58.04, Y 15.22, Z 16.0, A 0, B 90, C 0} C_DIS
LIN {X -58.28, Y 14.17, Z 16.0, A 0, B 90, C 0} C_DIS
LIN {X -58.89, Y 11.47, Z 16.0, A 0, B 90, C 0} C_DIS
LIN {X -59.07, Y 10.41, Z 16.0, A 0, B 90, C 0} C_DIS
LIN {X -59.51, Y 7.67, Z 16.0, A 0, B 90, C 0} C_DIS
LIN {X -59.61, Y 6.6, Z 16.0, A 0, B 90, C 0} C_DIS
LIN {X -59.88, Y 3.84, Z 16.0, A 0, B 90, C 0} C_DIS
LIN {X -59.91, Y 2.77, Z 16.0, A 0, B 90, C 0} C_DIS
LIN {X -60.0, Y -0.0, Z 16.0, A 0, B 90, C 0} C_DIS
LIN {X -59.97, Y -1.08, Z 16.0, A 0, B 90, C 0} C_DIS
LIN {X -59.88, Y -3.84, Z 16.0, A 0, B 90, C 0} C_DIS
LIN {X -59.77, Y -4.92, Z 16.0, A 0, B 90, C 0} C_DIS
LIN {X -59.51, Y -7.67, Z 16.0, A 0, B 90, C 0} C_DIS
LIN {X -59.34, Y -8.74, Z 16.0, A 0, B 90, C 0} C_DIS
LIN {X -58.89, Y -11.47, Z 16.0, A 0, B 90, C 0} C_DIS
LIN {X -58.65, Y -12.52, Z 16.0, A 0, B 90, C 0} C_DIS
LIN {X -58.04, Y -15.22, Z 16.0, A 0, B 90, C 0} C_DIS
LIN {X -57.73, Y -16.25, Z 16.0, A 0, B 90, C 0} C_DIS
LIN {X -56.94, Y -18.91, Z 16.0, A 0, B 90, C 0} C_DIS
LIN {X -56.57, Y -19.92, Z 16.0, A 0, B 90, C 0} C_DIS
LIN {X -55.62, Y -22.52, Z 16.0, A 0, B 90, C 0} C_DIS
LIN {X -55.18, Y -23.5, Z 16.0, A 0, B 90, C 0} C_DIS
LIN {X -54.06, Y -26.03, Z 16.0, A 0, B 90, C 0} C_DIS
LIN {X -53.56, Y -26.99, Z 16.0, A 0, B 90, C 0} C_DIS
LIN {X -52.28, Y -29.44, Z 16.0, A 0, B 90, C 0} C_DIS
LIN {X -51.72, Y -30.36, Z 16.0, A 0, B 90, C 0} C_DIS
LIN {X -50.29, Y -32.73, Z 16.0, A 0, B 90, C 0} C_DIS
LIN {X -49.67, Y -33.62, Z 16.0, A 0, B 90, C 0} C_DIS
LIN {X -48.08, Y -35.89, Z 16.0, A 0, B 90, C 0} C_DIS
LIN {X -47.41, Y -36.73, Z 16.0, A 0, B 90, C 0} C_DIS
LIN {X -45.69, Y -38.89, Z 16.0, A 0, B 90, C 0} C_DIS
LIN {X -44.96, Y -39.69, Z 16.0, A 0, B 90, C 0} C_DIS
LIN {X -43.1, Y -41.74, Z 16.0, A 0, B 90, C 0} C_DIS
LIN {X -42.33, Y -42.49, Z 16.0, A 0, B 90, C 0} C_DIS
LIN {X -40.34, Y -44.42, Z 16.0, A 0, B 90, C 0} C_DIS
LIN {X -39.52, Y -45.11, Z 16.0, A 0, B 90, C 0} C_DIS
LIN {X -37.41, Y -46.91, Z 16.0, A 0, B 90, C 0} C_DIS
LIN {X -36.55, Y -47.55, Z 16.0, A 0, B 90, C 0} C_DIS
$OUT[1] = FALSE

; END LAYER 7
LIN {X -34.33, Y -49.21, Z 16.0, A 0, B 90, C 0} C_DIS
WAIT SEC 3
LIN {X -34.33, Y -49.21, Z 18.0, A 0, B 90, C 0} C_DIS
$OUT[1] = TRUE
WAIT SEC 0.8
LIN {X -34.33, Y -49.21, Z 18.0, A 0, B 90, C 0} C_DIS
LIN {X -34.33, Y -49.21, Z 18.0, A 0, B 90, C 0} C_DIS
LIN {X -33.3, Y -49.88, Z 18.0, A 0, B 90, C 0} C_DIS
LIN {X -31.1, Y -51.31, Z 18.0, A 0, B 90, C 0} C_DIS
LIN {X -30.03, Y -51.91, Z 18.0, A 0, B 90, C 0} C_DIS
LIN {X -27.75, Y -53.2, Z 18.0, A 0, B 90, C 0} C_DIS
LIN {X -26.64, Y -53.73, Z 18.0, A 0, B 90, C 0} C_DIS
LIN {X -24.29, Y -54.86, Z 18.0, A 0, B 90, C 0} C_DIS
LIN {X -23.15, Y -55.33, Z 18.0, A 0, B 90, C 0} C_DIS
LIN {X -20.72, Y -56.31, Z 18.0, A 0, B 90, C 0} C_DIS
LIN {X -19.55, Y -56.7, Z 18.0, A 0, B 90, C 0} C_DIS
LIN {X -17.07, Y -57.52, Z 18.0, A 0, B 90, C 0} C_DIS
LIN {X -15.88, Y -57.83, Z 18.0, A 0, B 90, C 0} C_DIS
LIN {X -13.35, Y -58.5, Z 18.0, A 0, B 90, C 0} C_DIS
LIN {X -12.14, Y -58.73, Z 18.0, A 0, B 90, C 0} C_DIS
LIN {X -9.58, Y -59.23, Z 18.0, A 0, B 90, C 0} C_DIS
LIN {X -8.36, Y -59.39, Z 18.0, A 0, B 90, C 0} C_DIS
LIN {X -5.76, Y -59.72, Z 18.0, A 0, B 90, C 0} C_DIS
LIN {X -4.53, Y -59.8, Z 18.0, A 0, B 90, C 0} C_DIS
LIN {X -1.92, Y -59.97, Z 18.0, A 0, B 90, C 0} C_DIS
LIN {X -0.69, Y -59.97, Z 18.0, A 0, B 90, C 0} C_DIS
LIN {X 1.92, Y -59.97, Z 18.0, A 0, B 90, C 0} C_DIS
LIN {X 3.15, Y -59.89, Z 18.0, A 0, B 90, C 0} C_DIS
LIN {X 5.76, Y -59.72, Z 18.0, A 0, B 90, C 0} C_DIS
LIN {X 6.98, Y -59.57, Z 18.0, A 0, B 90, C 0} C_DIS
LIN {X 9.58, Y -59.23, Z 18.0, A 0, B 90, C 0} C_DIS
LIN {X 10.78, Y -59.0, Z 18.0, A 0, B 90, C 0} C_DIS
LIN {X 13.35, Y -58.5, Z 18.0, A 0, B 90, C 0} C_DIS
LIN {X 14.54, Y -58.18, Z 18.0, A 0, B 90, C 0} C_DIS
LIN {X 17.07, Y -57.52, Z 18.0, A 0, B 90, C 0} C_DIS
LIN {X 18.24, Y -57.13, Z 18.0, A 0, B 90, C 0} C_DIS
LIN {X 20.72, Y -56.31, Z 18.0, A 0, B 90, C 0} C_DIS
LIN {X 21.86, Y -55.85, Z 18.0, A 0, B 90, C 0} C_DIS
LIN {X 24.29, Y -54.86, Z 18.0, A 0, B 90, C 0} C_DIS
LIN {X 25.4, Y -54.33, Z 18.0, A 0, B 90, C 0} C_DIS
LIN {X 27.75, Y -53.2, Z 18.0, A 0, B 90, C 0} C_DIS
LIN {X 28.82, Y -52.59, Z 18.0, A 0, B 90, C 0} C_DIS
LIN {X 31.1, Y -51.31, Z 18.0, A 0, B 90, C 0} C_DIS
LIN {X 32.14, Y -50.64, Z 18.0, A 0, B 90, C 0} C_DIS
LIN {X 34.33, Y -49.21, Z 18.0, A 0, B 90, C 0} C_DIS
LIN {X 35.31, Y -48.47, Z 18.0, A 0, B 90, C 0} C_DIS
LIN {X 37.41, Y -46.91, Z 18.0, A 0, B 90, C 0} C_DIS
LIN {X 38.35, Y -46.11, Z 18.0, A 0, B 90, C 0} C_DIS
LIN {X 40.34, Y -44.42, Z 18.0, A 0, B 90, C 0} C_DIS
LIN {X 41.22, Y -43.56, Z 18.0, A 0, B 90, C 0} C_DIS
LIN {X 43.1, Y -41.74, Z 18.0, A 0, B 90, C 0} C_DIS
LIN {X 43.93, Y -40.83, Z 18.0, A 0, B 90, C 0} C_DIS
LIN {X 45.69, Y -38.89, Z 18.0, A 0, B 90, C 0} C_DIS
LIN {X 46.45, Y -37.93, Z 18.0, A 0, B 90, C 0} C_DIS
LIN {X 48.08, Y -35.89, Z 18.0, A 0, B 90, C 0} C_DIS
LIN {X 48.79, Y -34.88, Z 18.0, A 0, B 90, C 0} C_DIS
LIN {X 50.29, Y -32.73, Z 18.0, A 0, B 90, C 0} C_DIS
LIN {X 50.92, Y -31.68, Z 18.0, A 0, B 90, C 0} C_DIS
LIN {X 52.28, Y -29.44, Z 18.0, A 0, B 90, C 0} C_DIS
LIN {X 52.85, Y -28.35, Z 18.0, A 0, B 90, C 0} C_DIS
LIN {X 54.06, Y -26.03, Z 18.0, A 0, B 90, C 0} C_DIS
LIN {X 54.56, Y -24.91, Z 18.0, A 0, B 90, C 0} C_DIS
LIN {X 55.62, Y -22.52, Z 18.0, A 0, B 90, C 0} C_DIS
LIN {X 56.04, Y -21.36, Z 18.0, A 0, B 90, C 0} C_DIS
LIN {X 56.94, Y -18.91, Z 18.0, A 0, B 90, C 0} C_DIS
LIN {X 57.29, Y -17.73, Z 18.0, A 0, B 90, C 0} C_DIS
LIN {X 58.04, Y -15.22, Z 18.0, A 0, B 90, C 0} C_DIS
LIN {X 58.31, Y -14.02, Z 18.0, A 0, B 90, C 0} C_DIS
LIN {X 58.89, Y -11.47, Z 18.0, A 0, B 90, C 0} C_DIS
LIN {X 59.09, Y -10.25, Z 18.0, A 0, B 90, C 0} C_DIS
LIN {X 59.51, Y -7.67, Z 18.0, A 0, B 90, C 0} C_DIS
LIN {X 59.63, Y -6.45, Z 18.0, A 0, B 90, C 0} C_DIS
LIN {X 59.88, Y -3.84, Z 18.0, A 0, B 90, C 0} C_DIS
LIN {X 59.92, Y -2.61, Z 18.0, A 0, B 90, C 0} C_DIS
LIN {X 60.0, Y -0.0, Z 18.0, A 0, B 90, C 0} C_DIS
LIN {X 59.96, Y 1.23, Z 18.0, A 0, B 90, C 0} C_DIS
LIN {X 59.88, Y 3.84, Z 18.0, A 0, B 90, C 0} C_DIS
LIN {X 59.76, Y 5.07, Z 18.0, A 0, B 90, C 0} C_DIS
LIN {X 59.51, Y 7.67, Z 18.0, A 0, B 90, C 0} C_DIS
LIN {X 59.31, Y 8.89, Z 18.0, A 0, B 90, C 0} C_DIS
LIN {X 58.89, Y 11.47, Z 18.0, A 0, B 90, C 0} C_DIS
LIN {X 58.62, Y 12.67, Z 18.0, A 0, B 90, C 0} C_DIS
LIN {X 58.04, Y 15.22, Z 18.0, A 0, B 90, C 0} C_DIS
LIN {X 57.69, Y 16.4, Z 18.0, A 0, B 90, C 0} C_DIS
LIN {X 56.94, Y 18.91, Z 18.0, A 0, B 90, C 0} C_DIS
LIN {X 56.52, Y 20.06, Z 18.0, A 0, B 90, C 0} C_DIS
LIN {X 55.62, Y 22.52, Z 18.0, A 0, B 90, C 0} C_DIS
LIN {X 55.12, Y 23.64, Z 18.0, A 0, B 90, C 0} C_DIS
LIN {X 54.06, Y 26.03, Z 18.0, A 0, B 90, C 0} C_DIS
LIN {X 53.49, Y 27.12, Z 18.0, A 0, B 90, C 0} C_DIS
LIN {X 52.28, Y 29.44, Z 18.0, A 0, B 90, C 0} C_DIS
LIN {X 51.64, Y 30.5, Z 18.0, A 0, B 90, C 0} C_DIS
LIN {X 50.29, Y 32.73, Z 18.0, A 0, B 90, C 0} C_DIS
LIN {X 49.58, Y 33.74, Z 18.0, A 0, B 90, C 0} C_DIS
LIN {X 48.08, Y 35.89, Z 18.0, A 0, B 90, C 0} C_DIS
LIN {X 47.32, Y 36.85, Z 18.0, A 0, B 90, C 0} C_DIS
LIN {X 45.69, Y 38.89, Z 18.0, A 0, B 90, C 0} C_DIS
LIN {X 44.86, Y 39.8, Z 18.0, A 0, B 90, C 0} C_DIS
LIN {X 43.1, Y 41.74, Z 18.0, A 0, B 90, C 0} C_DIS
LIN {X 42.22, Y 42.6, Z 18.0, A 0, B 90, C 0} C_DIS
LIN {X 40.34, Y 44.42, Z 18.0, A 0, B 90, C 0} C_DIS
LIN {X 39.4, Y 45.21, Z 18.0, A 0, B 90, C 0} C_DIS
LIN {X 37.41, Y 46.91, Z 18.0, A 0, B 90, C 0} C_DIS
LIN {X 36.42, Y 47.65, Z 18.0, A 0, B 90, C 0} C_DIS
LIN {X 34.33, Y 49.21, Z 18.0, A 0, B 90, C 0} C_DIS
LIN {X 33.3, Y 49.88, Z 18.0, A 0, B 90, C 0} C_DIS
LIN {X 31.1, Y 51.31, Z 18.0, A 0, B 90, C 0} C_DIS
LIN {X 30.03, Y 51.91, Z 18.0, A 0, B 90, C 0} C_DIS
LIN {X 27.75, Y 53.2, Z 18.0, A 0, B 90, C 0} C_DIS
LIN {X 26.64, Y 53.73, Z 18.0, A 0, B 90, C 0} C_DIS
LIN {X 24.29, Y 54.86, Z 18.0, A 0, B 90, C 0} C_DIS
LIN {X 23.15, Y 55.33, Z 18.0, A 0, B 90, C 0} C_DIS
LIN {X 20.72, Y 56.31, Z 18.0, A 0, B 90, C 0} C_DIS
LIN {X 19.55, Y 56.7, Z 18.0, A 0, B 90, C 0} C_DIS
LIN {X 17.07, Y 57.52, Z 18.0, A 0, B 90, C 0} C_DIS
LIN {X 15.88, Y 57.83, Z 18.0, A 0, B 90, C 0} C_DIS
LIN {X 13.35, Y 58.5, Z 18.0, A 0, B 90, C 0} C_DIS
LIN {X 12.14, Y 58.73, Z 18.0, A 0, B 90, C 0} C_DIS
LIN {X 9.58, Y 59.23, Z 18.0, A 0, B 90, C 0} C_DIS
LIN {X 8.36, Y 59.39, Z 18.0, A 0, B 90, C 0} C_DIS
LIN {X 5.76, Y 59.72, Z 18.0, A 0, B 90, C 0} C_DIS
LIN {X 4.53, Y 59.8, Z 18.0, A 0, B 90, C 0} C_DIS
LIN {X 1.92, Y 59.97, Z 18.0, A 0, B 90, C 0} C_DIS
LIN {X 0.69, Y 59.97, Z 18.0, A 0, B 90, C 0} C_DIS
LIN {X -1.92, Y 59.97, Z 18.0, A 0, B 90, C 0} C_DIS
LIN {X -3.15, Y 59.89, Z 18.0, A 0, B 90, C 0} C_DIS
LIN {X -5.76, Y 59.72, Z 18.0, A 0, B 90, C 0} C_DIS
LIN {X -6.98, Y 59.57, Z 18.0, A 0, B 90, C 0} C_DIS
LIN {X -9.58, Y 59.23, Z 18.0, A 0, B 90, C 0} C_DIS
LIN {X -10.78, Y 59.0, Z 18.0, A 0, B 90, C 0} C_DIS
LIN {X -13.35, Y 58.5, Z 18.0, A 0, B 90, C 0} C_DIS
LIN {X -14.54, Y 58.18, Z 18.0, A 0, B 90, C 0} C_DIS
LIN {X -17.07, Y 57.52, Z 18.0, A 0, B 90, C 0} C_DIS
LIN {X -18.24, Y 57.13, Z 18.0, A 0, B 90, C 0} C_DIS
LIN {X -20.72, Y 56.31, Z 18.0, A 0, B 90, C 0} C_DIS
LIN {X -21.86, Y 55.85, Z 18.0, A 0, B 90, C 0} C_DIS
LIN {X -24.29, Y 54.86, Z 18.0, A 0, B 90, C 0} C_DIS
LIN {X -25.4, Y 54.33, Z 18.0, A 0, B 90, C 0} C_DIS
LIN {X -27.75, Y 53.2, Z 18.0, A 0, B 90, C 0} C_DIS
LIN {X -28.82, Y 52.59, Z 18.0, A 0, B 90, C 0} C_DIS
LIN {X -31.1, Y 51.31, Z 18.0, A 0, B 90, C 0} C_DIS
LIN {X -32.14, Y 50.64, Z 18.0, A 0, B 90, C 0} C_DIS
LIN {X -34.33, Y 49.21, Z 18.0, A 0, B 90, C 0} C_DIS
LIN {X -35.31, Y 48.47, Z 18.0, A 0, B 90, C 0} C_DIS
LIN {X -37.41, Y 46.91, Z 18.0, A 0, B 90, C 0} C_DIS
LIN {X -38.35, Y 46.11, Z 18.0, A 0, B 90, C 0} C_DIS
LIN {X -40.34, Y 44.42, Z 18.0, A 0, B 90, C 0} C_DIS
LIN {X -41.22, Y 43.56, Z 18.0, A 0, B 90, C 0} C_DIS
LIN {X -43.1, Y 41.74, Z 18.0, A 0, B 90, C 0} C_DIS
LIN {X -43.93, Y 40.83, Z 18.0, A 0, B 90, C 0} C_DIS
LIN {X -45.69, Y 38.89, Z 18.0, A 0, B 90, C 0} C_DIS
LIN {X -46.45, Y 37.93, Z 18.0, A 0, B 90, C 0} C_DIS
LIN {X -48.08, Y 35.89, Z 18.0, A 0, B 90, C 0} C_DIS
LIN {X -48.79, Y 34.88, Z 18.0, A 0, B 90, C 0} C_DIS
LIN {X -50.29, Y 32.73, Z 18.0, A 0, B 90, C 0} C_DIS
LIN {X -50.92, Y 31.68, Z 18.0, A 0, B 90, C 0} C_DIS
LIN {X -52.28, Y 29.44, Z 18.0, A 0, B 90, C 0} C_DIS
LIN {X -52.85, Y 28.35, Z 18.0, A 0, B 90, C 0} C_DIS
LIN {X -54.06, Y 26.03, Z 18.0, A 0, B 90, C 0} C_DIS
LIN {X -54.56, Y 24.91, Z 18.0, A 0, B 90, C 0} C_DIS
LIN {X -55.62, Y 22.52, Z 18.0, A 0, B 90, C 0} C_DIS
LIN {X -56.04, Y 21.36, Z 18.0, A 0, B 90, C 0} C_DIS
LIN {X -56.94, Y 18.91, Z 18.0, A 0, B 90, C 0} C_DIS
LIN {X -57.29, Y 17.73, Z 18.0, A 0, B 90, C 0} C_DIS
LIN {X -58.04, Y 15.22, Z 18.0, A 0, B 90, C 0} C_DIS
LIN {X -58.31, Y 14.02, Z 18.0, A 0, B 90, C 0} C_DIS
LIN {X -58.89, Y 11.47, Z 18.0, A 0, B 90, C 0} C_DIS
LIN {X -59.09, Y 10.25, Z 18.0, A 0, B 90, C 0} C_DIS
LIN {X -59.51, Y 7.67, Z 18.0, A 0, B 90, C 0} C_DIS
LIN {X -59.63, Y 6.45, Z 18.0, A 0, B 90, C 0} C_DIS
LIN {X -59.88, Y 3.84, Z 18.0, A 0, B 90, C 0} C_DIS
LIN {X -59.92, Y 2.61, Z 18.0, A 0, B 90, C 0} C_DIS
LIN {X -60.0, Y -0.0, Z 18.0, A 0, B 90, C 0} C_DIS
LIN {X -59.96, Y -1.23, Z 18.0, A 0, B 90, C 0} C_DIS
LIN {X -59.88, Y -3.84, Z 18.0, A 0, B 90, C 0} C_DIS
LIN {X -59.76, Y -5.07, Z 18.0, A 0, B 90, C 0} C_DIS
LIN {X -59.51, Y -7.67, Z 18.0, A 0, B 90, C 0} C_DIS
LIN {X -59.31, Y -8.89, Z 18.0, A 0, B 90, C 0} C_DIS
LIN {X -58.89, Y -11.47, Z 18.0, A 0, B 90, C 0} C_DIS
LIN {X -58.62, Y -12.67, Z 18.0, A 0, B 90, C 0} C_DIS
LIN {X -58.04, Y -15.22, Z 18.0, A 0, B 90, C 0} C_DIS
LIN {X -57.69, Y -16.4, Z 18.0, A 0, B 90, C 0} C_DIS
LIN {X -56.94, Y -18.91, Z 18.0, A 0, B 90, C 0} C_DIS
LIN {X -56.52, Y -20.06, Z 18.0, A 0, B 90, C 0} C_DIS
LIN {X -55.62, Y -22.52, Z 18.0, A 0, B 90, C 0} C_DIS
LIN {X -55.12, Y -23.64, Z 18.0, A 0, B 90, C 0} C_DIS
LIN {X -54.06, Y -26.03, Z 18.0, A 0, B 90, C 0} C_DIS
LIN {X -53.49, Y -27.12, Z 18.0, A 0, B 90, C 0} C_DIS
LIN {X -52.28, Y -29.44, Z 18.0, A 0, B 90, C 0} C_DIS
LIN {X -51.64, Y -30.5, Z 18.0, A 0, B 90, C 0} C_DIS
LIN {X -50.29, Y -32.73, Z 18.0, A 0, B 90, C 0} C_DIS
LIN {X -49.58, Y -33.74, Z 18.0, A 0, B 90, C 0} C_DIS
LIN {X -48.08, Y -35.89, Z 18.0, A 0, B 90, C 0} C_DIS
LIN {X -47.32, Y -36.85, Z 18.0, A 0, B 90, C 0} C_DIS
LIN {X -45.69, Y -38.89, Z 18.0, A 0, B 90, C 0} C_DIS
LIN {X -44.86, Y -39.8, Z 18.0, A 0, B 90, C 0} C_DIS
LIN {X -43.1, Y -41.74, Z 18.0, A 0, B 90, C 0} C_DIS
LIN {X -42.22, Y -42.6, Z 18.0, A 0, B 90, C 0} C_DIS
LIN {X -40.34, Y -44.42, Z 18.0, A 0, B 90, C 0} C_DIS
LIN {X -39.4, Y -45.21, Z 18.0, A 0, B 90, C 0} C_DIS
LIN {X -37.41, Y -46.91, Z 18.0, A 0, B 90, C 0} C_DIS
LIN {X -36.42, Y -47.65, Z 18.0, A 0, B 90, C 0} C_DIS
$OUT[1] = FALSE

